LIN {X 0,Y 157.463,Z 192.851,A -85,B 0,C 180,E1 -23744.468,E2 -23744.468} C_VEL
LIN {X 0,Y 157.689,Z 192.84,A -85,B 0,C 180,E1 -23749.732,E2 -23749.732} C_VEL
LIN {X 0,Y 157.768,Z 192.832,A -85,B 0,C 180,E1 -23752.321,E2 -23752.321} C_VEL
LIN {X 0,Y 158.258,Z 192.764,A -85,B 0,C 180,E1 -23760.001,E2 -23760.001} C_VEL
LIN {X 0,Y 157.765,Z 192.822,A -85,B 0,C 180,E1 -23767.681,E2 -23767.681} C_VEL
LIN {X 0,Y 157.639,Z 192.844,A -85,B 0,C 180,E1 -23771.239,E2 -23771.239} C_VEL
LIN {X 0,Y 157.481,Z 192.867,A -85,B 0,C 180,E1 -23775.533,E2 -23775.533} C_VEL
LIN {X 0,Y 157.417,Z 192.875,A -85,B 0,C 180,E1 -23780.928,E2 -23780.928} C_VEL
LIN {X 0,Y 157.316,Z 192.89,A -85,B 0,C 180,E1 -23786.686,E2 -23786.686} C_VEL
LIN {X 0,Y 157.394,Z 192.935,A -85,B 0,C 180,E1 -23790.721,E2 -23790.721} C_VEL
LIN {X 0,Y 158.004,Z 196.792,A -85,B 0,C 180,E1 -23796.809,E2 -23796.809} C_VEL
LIN {X 0,Y 158.869,Z 201.219,A -85,B 0,C 180,E1 -23803.291,E2 -23803.291} C_VEL
LIN {X 0,Y 159.673,Z 205.204,A -85,B 0,C 180,E1 -23808.683,E2 -23808.683} C_VEL
LIN {X 0,Y 159.874,Z 206.674,A -85,B 0,C 180,E1 -23810.49,E2 -23810.49} C_VEL
LIN {X 0,Y 162.118,Z 215.988,A -85,B 0,C 180,E1 -23811.767,E2 -23811.767} C_VEL
LIN {X 0,Y 163.887,Z 229.522,A -85,B 0,C 180,E1 -23813.781,E2 -23813.781} C_VEL
LIN {X 0,Y 164.833,Z 241.541,A -85,B 0,C 180,E1 -23815.928,E2 -23815.928} C_VEL
LIN {X 0,Y 165.292,Z 252.413,A -85,B 0,C 180,E1 -23818.254,E2 -23818.254} C_VEL
LIN {X 0,Y 165.267,Z 263.527,A -85,B 0,C 180,E1 -23821.072,E2 -23821.072} C_VEL
LIN {X 0,Y 164.96,Z 269.314,A -85,B 0,C 180,E1 -23822.743,E2 -23822.743} C_VEL
LIN {X 0,Y 162.355,Z 278.226,A -85,B 0,C 180,E1 -23825.6,E2 -23825.6} C_VEL
LIN {X 0,Y 159.702,Z 287.461,A -85,B 0,C 180,E1 -23829.387,E2 -23829.387} C_VEL
LIN {X 0,Y 157.604,Z 294.658,A -85,B 0,C 180,E1 -23833.151,E2 -23833.151} C_VEL
LIN {X 0,Y 156.231,Z 300.428,A -85,B 0,C 180,E1 -23837.002,E2 -23837.002} C_VEL
LIN {X 0,Y 155.46,Z 304.944,A -85,B 0,C 180,E1 -23840.896,E2 -23840.896} C_VEL
LIN {X 0,Y 155.217,Z 308.458,A -85,B 0,C 180,E1 -23844.971,E2 -23844.971} C_VEL
LIN {X 0,Y 155.265,Z 310.005,A -85,B 0,C 180,E1 -23847.406,E2 -23847.406} C_VEL
LIN {X 0,Y 155.288,Z 311.229,A -85,B 0,C 180,E1 -23850,E2 -23850} C_VEL
LIN {X 0,Y 155.038,Z 312.3,A -85,B 0,C 180,E1 -23854.211,E2 -23854.211} C_VEL
LIN {X 0,Y 155.096,Z 312.412,A -85,B 0,C 180,E1 -23857.814,E2 -23857.814} C_VEL
LIN {X 0,Y 156.1,Z 311.257,A -85,B 0,C 180,E1 -23863.01,E2 -23863.01} C_VEL
LIN {X 0,Y 158.288,Z 308.643,A -85,B 0,C 180,E1 -23868.108,E2 -23868.108} C_VEL
LIN {X 0,Y 160.859,Z 305.623,A -85,B 0,C 180,E1 -23871.801,E2 -23871.801} C_VEL
LIN {X 0,Y 164.073,Z 301.657,A -85,B 0,C 180,E1 -23875.363,E2 -23875.363} C_VEL
LIN {X 0,Y 167.812,Z 296.682,A -85,B 0,C 180,E1 -23878.792,E2 -23878.792} C_VEL
LIN {X 0,Y 173.037,Z 289.457,A -85,B 0,C 180,E1 -23882.559,E2 -23882.559} C_VEL
LIN {X 0,Y 177.266,Z 283.144,A -85,B 0,C 180,E1 -23885.092,E2 -23885.092} C_VEL
LIN {X 0,Y 180.54,Z 275.915,A -85,B 0,C 180,E1 -23887.815,E2 -23887.815} C_VEL
LIN {X 0,Y 183.154,Z 267.778,A -85,B 0,C 180,E1 -23890.718,E2 -23890.718} C_VEL
LIN {X 0,Y 184.392,Z 262.401,A -85,B 0,C 180,E1 -23892.591,E2 -23892.591} C_VEL
LIN {X 0,Y 184.603,Z 260.007,A -85,B 0,C 180,E1 -23893.557,E2 -23893.557} C_VEL
LIN {X 0,Y 184.01,Z 257.051,A -85,B 0,C 180,E1 -23895.144,E2 -23895.144} C_VEL
LIN {X 0,Y 181.779,Z 253.248,A -85,B 0,C 180,E1 -23897.989,E2 -23897.989} C_VEL
LIN {X 0,Y 180.006,Z 250.364,A -85,B 0,C 180,E1 -23900.365,E2 -23900.365} C_VEL
LIN {X 0,Y 179.466,Z 248.695,A -85,B 0,C 180,E1 -23901.549,E2 -23901.549} C_VEL
LIN {X 0,Y 178.396,Z 243.679,A -85,B 0,C 180,E1 -23905.164,E2 -23905.164} C_VEL
LIN {X 0,Y 177.445,Z 239.467,A -85,B 0,C 180,E1 -23909.009,E2 -23909.009} C_VEL
LIN {X 0,Y 176.338,Z 236.354,A -85,B 0,C 180,E1 -23913.996,E2 -23913.996} C_VEL
LIN {X 0,Y 176.156,Z 235.271,A -85,B 0,C 180,E1 -23916.582,E2 -23916.582} C_VEL
LIN {X 0,Y 176.198,Z 234.757,A -85,B 0,C 180,E1 -23918.961,E2 -23918.961} C_VEL
LIN {X 0,Y 176.858,Z 234.904,A -85,B 0,C 180,E1 -23923.848,E2 -23923.848} C_VEL
LIN {X 0,Y 177.644,Z 235.267,A -85,B 0,C 180,E1 -23926.267,E2 -23926.267} C_VEL
LIN {X 0,Y 178.999,Z 238.295,A -85,B 0,C 180,E1 -23930.963,E2 -23930.963} C_VEL
LIN {X 0,Y 180.79,Z 242.663,A -85,B 0,C 180,E1 -23935.54,E2 -23935.54} C_VEL
LIN {X 0,Y 181.708,Z 247.304,A -85,B 0,C 180,E1 -23938.891,E2 -23938.891} C_VEL
LIN {X 0,Y 182.129,Z 251.884,A -85,B 0,C 180,E1 -23941.657,E2 -23941.657} C_VEL
LIN {X 0,Y 181.604,Z 258.398,A -85,B 0,C 180,E1 -23944.994,E2 -23944.994} C_VEL
LIN {X 0,Y 181.219,Z 260.675,A -85,B 0,C 180,E1 -23946.121,E2 -23946.121} C_VEL
LIN {X 0,Y 180.563,Z 262.357,A -85,B 0,C 180,E1 -23946.785,E2 -23946.785} C_VEL
LIN {X 0,Y 174.841,Z 270.868,A -85,B 0,C 180,E1 -23949.725,E2 -23949.725} C_VEL
LIN {X 0,Y 169.025,Z 278.432,A -85,B 0,C 180,E1 -23953.184,E2 -23953.184} C_VEL
LIN {X 0,Y 163.924,Z 284.316,A -85,B 0,C 180,E1 -23956.82,E2 -23956.82} C_VEL
LIN {X 0,Y 159.457,Z 288.794,A -85,B 0,C 180,E1 -23960.645,E2 -23960.645} C_VEL
LIN {X 0,Y 155.341,Z 292.384,A -85,B 0,C 180,E1 -23965.195,E2 -23965.195} C_VEL
LIN {X 0,Y 152.671,Z 294.266,A -85,B 0,C 180,E1 -23968.997,E2 -23968.997} C_VEL
LIN {X 0,Y 150.028,Z 295.433,A -85,B 0,C 180,E1 -23974.202,E2 -23974.202} C_VEL
LIN {X 0,Y 148.835,Z 295.324,A -85,B 0,C 180,E1 -23977.867,E2 -23977.867} C_VEL
LIN {X 0,Y 148.082,Z 294.5,A -85,B 0,C 180,E1 -23981.638,E2 -23981.638} C_VEL
LIN {X 0,Y 147.8,Z 292.89,A -85,B 0,C 180,E1 -23985.499,E2 -23985.499} C_VEL
LIN {X 0,Y 148.195,Z 289.33,A -85,B 0,C 180,E1 -23990.732,E2 -23990.732} C_VEL
LIN {X 0,Y 149.299,Z 284.523,A -85,B 0,C 180,E1 -23995.605,E2 -23995.605} C_VEL
LIN {X 0,Y 150.77,Z 278.971,A -85,B 0,C 180,E1 -23999.803,E2 -23999.803} C_VEL
LIN {X 0,Y 152.869,Z 271.595,A -85,B 0,C 180,E1 -24004.102,E2 -24004.102} C_VEL
LIN {X 0,Y 155.593,Z 262.734,A -85,B 0,C 180,E1 -24008.121,E2 -24008.121} C_VEL
LIN {X 0,Y 158.457,Z 252.842,A -85,B 0,C 180,E1 -24011.599,E2 -24011.599} C_VEL
LIN {X 0,Y 161.225,Z 242.566,A -85,B 0,C 180,E1 -24014.457,E2 -24014.457} C_VEL
LIN {X 0,Y 162.267,Z 237.854,A -85,B 0,C 180,E1 -24015.579,E2 -24015.579} C_VEL
LIN {X 0,Y 160.82,Z 227.521,A -85,B 0,C 180,E1 -24018.241,E2 -24018.241} C_VEL
LIN {X 0,Y 158.624,Z 216.159,A -85,B 0,C 180,E1 -24020.807,E2 -24020.807} C_VEL
LIN {X 0,Y 155.818,Z 206.445,A -85,B 0,C 180,E1 -24022.867,E2 -24022.867} C_VEL
LIN {X 0,Y 151.984,Z 197.063,A -85,B 0,C 180,E1 -24024.859,E2 -24024.859} C_VEL
LIN {X 0,Y 150.781,Z 194.317,A -85,B 0,C 180,E1 -24025.405,E2 -24025.405} C_VEL
LIN {X 0,Y 150.684,Z 193.719,A -85,B 0,C 180,E1 -24025.569,E2 -24025.569} C_VEL
LIN {X 0,Y 151.216,Z 193.647,A -85,B 0,C 180,E1 -24030,E2 -24030} C_VEL
LIN {X 0,Y 150.76,Z 193.71,A -85,B 0,C 180,E1 -24038.039,E2 -24038.039} C_VEL
LIN {X 0,Y 150.632,Z 193.719,A -85,B 0,C 180,E1 -24041.546,E2 -24041.546} C_VEL
LIN {X 0,Y 150.394,Z 193.752,A -85,B 0,C 180,E1 -24046.283,E2 -24046.283} C_VEL
LIN {X 0,Y 150.387,Z 193.756,A -85,B 0,C 180,E1 -24050.831,E2 -24050.831} C_VEL
LIN {X 0,Y 150.241,Z 193.761,A -85,B 0,C 180,E1 -24057.282,E2 -24057.282} C_VEL
LIN {X 0,Y 150.211,Z 193.775,A -85,B 0,C 180,E1 -24062.632,E2 -24062.632} C_VEL
LIN {X 0,Y 150.169,Z 193.766,A -85,B 0,C 180,E1 -24067.474,E2 -24067.474} C_VEL
LIN {X 0,Y 150.147,Z 193.782,A -85,B 0,C 180,E1 -24071.505,E2 -24071.505} C_VEL
LIN {X 0,Y 150.123,Z 193.777,A -85,B 0,C 180,E1 -24075.396,E2 -24075.396} C_VEL
LIN {X 0,Y 150.147,Z 193.764,A -85,B 0,C 180,E1 -24079.059,E2 -24079.059} C_VEL
LIN {X 0,Y 150.177,Z 193.775,A -85,B 0,C 180,E1 -24082.709,E2 -24082.709} C_VEL
LIN {X 0,Y 150.212,Z 193.768,A -85,B 0,C 180,E1 -24087.369,E2 -24087.369} C_VEL
LIN {X 0,Y 150.242,Z 193.753,A -85,B 0,C 180,E1 -24092.719,E2 -24092.719} C_VEL
LIN {X 0,Y 150.389,Z 193.749,A -85,B 0,C 180,E1 -24099.17,E2 -24099.17} C_VEL
LIN {X 0,Y 150.375,Z 193.735,A -85,B 0,C 180,E1 -24103.716,E2 -24103.716} C_VEL
LIN {X 0,Y 150.611,Z 193.721,A -85,B 0,C 180,E1 -24109.244,E2 -24109.244} C_VEL
LIN {X 0,Y 150.705,Z 193.713,A -85,B 0,C 180,E1 -24111.959,E2 -24111.959} C_VEL
LIN {X 0,Y 151.218,Z 193.64,A -85,B 0,C 180,E1 -24120.001,E2 -24120.001} C_VEL
LIN {X 0,Y 150.687,Z 193.701,A -85,B 0,C 180,E1 -24128.045,E2 -24128.045} C_VEL
LIN {X 0,Y 150.579,Z 193.724,A -85,B 0,C 180,E1 -24131.439,E2 -24131.439} C_VEL
LIN {X 0,Y 150.392,Z 193.746,A -85,B 0,C 180,E1 -24136.285,E2 -24136.285} C_VEL
LIN {X 0,Y 150.391,Z 193.75,A -85,B 0,C 180,E1 -24140.833,E2 -24140.833} C_VEL
LIN {X 0,Y 150.248,Z 193.772,A -85,B 0,C 180,E1 -24147.285,E2 -24147.285} C_VEL
LIN {X 0,Y 150.294,Z 193.83,A -85,B 0,C 180,E1 -24150.18,E2 -24150.18} C_VEL
LIN {X 0,Y 150.639,Z 196.137,A -85,B 0,C 180,E1 -24154.047,E2 -24154.047} C_VEL
LIN {X 0,Y 151.081,Z 198.423,A -85,B 0,C 180,E1 -24157.74,E2 -24157.74} C_VEL
LIN {X 0,Y 151.903,Z 202.558,A -85,B 0,C 180,E1 -24163.949,E2 -24163.949} C_VEL
LIN {X 0,Y 152.673,Z 206.336,A -85,B 0,C 180,E1 -24169.059,E2 -24169.059} C_VEL
LIN {X 0,Y 153.739,Z 209.669,A -85,B 0,C 180,E1 -24169.566,E2 -24169.566} C_VEL
LIN {X 0,Y 155.719,Z 217.222,A -85,B 0,C 180,E1 -24170.741,E2 -24170.741} C_VEL
LIN {X 0,Y 157.251,Z 229.909,A -85,B 0,C 180,E1 -24172.739,E2 -24172.739} C_VEL
LIN {X 0,Y 158.108,Z 241.252,A -85,B 0,C 180,E1 -24174.895,E2 -24174.895} C_VEL
LIN {X 0,Y 158.475,Z 252.458,A -85,B 0,C 180,E1 -24177.418,E2 -24177.418} C_VEL
LIN {X 0,Y 158.385,Z 263.687,A -85,B 0,C 180,E1 -24180.42,E2 -24180.42} C_VEL
LIN {X 0,Y 158.044,Z 269.421,A -85,B 0,C 180,E1 -24182.166,E2 -24182.166} C_VEL
LIN {X 0,Y 155.213,Z 278.695,A -85,B 0,C 180,E1 -24185.328,E2 -24185.328} C_VEL
LIN {X 0,Y 152.622,Z 287.374,A -85,B 0,C 180,E1 -24189.092,E2 -24189.092} C_VEL
LIN {X 0,Y 150.504,Z 294.512,A -85,B 0,C 180,E1 -24193.032,E2 -24193.032} C_VEL
LIN {X 0,Y 149.303,Z 299.333,A -85,B 0,C 180,E1 -24196.388,E2 -24196.388} C_VEL
LIN {X 0,Y 148.458,Z 303.997,A -85,B 0,C 180,E1 -24200.463,E2 -24200.463} C_VEL
LIN {X 0,Y 148.143,Z 307.892,A -85,B 0,C 180,E1 -24205.052,E2 -24205.052} C_VEL
LIN {X 0,Y 148.183,Z 309.302,A -85,B 0,C 180,E1 -24207.282,E2 -24207.282} C_VEL
LIN {X 0,Y 148.226,Z 310.592,A -85,B 0,C 180,E1 -24210,E2 -24210} C_VEL
LIN {X 0,Y 147.977,Z 311.743,A -85,B 0,C 180,E1 -24214.137,E2 -24214.137} C_VEL
LIN {X 0,Y 148.036,Z 311.979,A -85,B 0,C 180,E1 -24218.189,E2 -24218.189} C_VEL
LIN {X 0,Y 148.467,Z 311.676,A -85,B 0,C 180,E1 -24220.915,E2 -24220.915} C_VEL
LIN {X 0,Y 150.123,Z 309.924,A -85,B 0,C 180,E1 -24226.314,E2 -24226.314} C_VEL
LIN {X 0,Y 153.299,Z 306.7,A -85,B 0,C 180,E1 -24231.516,E2 -24231.516} C_VEL
LIN {X 0,Y 156.451,Z 303.214,A -85,B 0,C 180,E1 -24235.262,E2 -24235.262} C_VEL
LIN {X 0,Y 160.239,Z 298.763,A -85,B 0,C 180,E1 -24238.846,E2 -24238.846} C_VEL
LIN {X 0,Y 165.431,Z 292.227,A -85,B 0,C 180,E1 -24242.797,E2 -24242.797} C_VEL
LIN {X 0,Y 170.716,Z 285.201,A -85,B 0,C 180,E1 -24245.92,E2 -24245.92} C_VEL
LIN {X 0,Y 174.343,Z 278.487,A -85,B 0,C 180,E1 -24248.67,E2 -24248.67} C_VEL
LIN {X 0,Y 177.251,Z 270.999,A -85,B 0,C 180,E1 -24251.548,E2 -24251.548} C_VEL
LIN {X 0,Y 179.318,Z 263.592,A -85,B 0,C 180,E1 -24254.298,E2 -24254.298} C_VEL
LIN {X 0,Y 180.404,Z 258.267,A -85,B 0,C 180,E1 -24256.313,E2 -24256.313} C_VEL
LIN {X 0,Y 180.532,Z 255.172,A -85,B 0,C 180,E1 -24257.703,E2 -24257.703} C_VEL
LIN {X 0,Y 179.466,Z 248.695,A -85,B 0,C 180,E1 -24261.549,E2 -24261.549} C_VEL
LIN {X 0,Y 178.564,Z 246.71,A -85,B 0,C 180,E1 -24263.301,E2 -24263.301} C_VEL
LIN {X 0,Y 177.18,Z 245.666,A -85,B 0,C 180,E1 -24265.131,E2 -24265.131} C_VEL
LIN {X 0,Y 173.518,Z 244.495,A -85,B 0,C 180,E1 -24270.247,E2 -24270.247} C_VEL
LIN {X 0,Y 173.088,Z 243.904,A -85,B 0,C 180,E1 -24271.56,E2 -24271.56} C_VEL
LIN {X 0,Y 172.619,Z 241.728,A -85,B 0,C 180,E1 -24275.974,E2 -24275.974} C_VEL
LIN {X 0,Y 172.701,Z 240.889,A -85,B 0,C 180,E1 -24279.388,E2 -24279.388} C_VEL
LIN {X 0,Y 173.866,Z 241.276,A -85,B 0,C 180,E1 -24285.963,E2 -24285.963} C_VEL
LIN {X 0,Y 174.98,Z 244.09,A -85,B 0,C 180,E1 -24290.754,E2 -24290.754} C_VEL
LIN {X 0,Y 176.319,Z 248.343,A -85,B 0,C 180,E1 -24295.426,E2 -24295.426} C_VEL
LIN {X 0,Y 176.829,Z 252.868,A -85,B 0,C 180,E1 -24298.86,E2 -24298.86} C_VEL
LIN {X 0,Y 176.825,Z 256.432,A -85,B 0,C 180,E1 -24301.138,E2 -24301.138} C_VEL
LIN {X 0,Y 175.838,Z 262.639,A -85,B 0,C 180,E1 -24304.584,E2 -24304.584} C_VEL
LIN {X 0,Y 175.509,Z 263.762,A -85,B 0,C 180,E1 -24305.168,E2 -24305.168} C_VEL
LIN {X 0,Y 170.267,Z 271.258,A -85,B 0,C 180,E1 -24307.845,E2 -24307.845} C_VEL
LIN {X 0,Y 164.664,Z 278.164,A -85,B 0,C 180,E1 -24310.986,E2 -24310.986} C_VEL
LIN {X 0,Y 159.568,Z 283.694,A -85,B 0,C 180,E1 -24314.309,E2 -24314.309} C_VEL
LIN {X 0,Y 154.119,Z 288.91,A -85,B 0,C 180,E1 -24318.614,E2 -24318.614} C_VEL
LIN {X 0,Y 149.289,Z 292.805,A -85,B 0,C 180,E1 -24323.586,E2 -24323.586} C_VEL
LIN {X 0,Y 145.486,Z 295.163,A -85,B 0,C 180,E1 -24328.884,E2 -24328.884} C_VEL
LIN {X 0,Y 143.17,Z 295.928,A -85,B 0,C 180,E1 -24333.434,E2 -24333.434} C_VEL
LIN {X 0,Y 141.796,Z 295.721,A -85,B 0,C 180,E1 -24337.53,E2 -24337.53} C_VEL
LIN {X 0,Y 140.981,Z 294.721,A -85,B 0,C 180,E1 -24341.602,E2 -24341.602} C_VEL
LIN {X 0,Y 140.698,Z 292.969,A -85,B 0,C 180,E1 -24345.627,E2 -24345.627} C_VEL
LIN {X 0,Y 141.18,Z 289.173,A -85,B 0,C 180,E1 -24351.236,E2 -24351.236} C_VEL
LIN {X 0,Y 142.094,Z 285.274,A -85,B 0,C 180,E1 -24355.309,E2 -24355.309} C_VEL
LIN {X 0,Y 143.619,Z 279.574,A -85,B 0,C 180,E1 -24359.895,E2 -24359.895} C_VEL
LIN {X 0,Y 145.721,Z 272.467,A -85,B 0,C 180,E1 -24364.274,E2 -24364.274} C_VEL
LIN {X 0,Y 148.334,Z 264.163,A -85,B 0,C 180,E1 -24368.28,E2 -24368.28} C_VEL
LIN {X 0,Y 151.104,Z 255.196,A -85,B 0,C 180,E1 -24371.702,E2 -24371.702} C_VEL
LIN {X 0,Y 154.096,Z 244.667,A -85,B 0,C 180,E1 -24374.857,E2 -24374.857} C_VEL
LIN {X 0,Y 155.494,Z 239.051,A -85,B 0,C 180,E1 -24376.273,E2 -24376.273} C_VEL
LIN {X 0,Y 154.078,Z 228.523,A -85,B 0,C 180,E1 -24379.154,E2 -24379.154} C_VEL
LIN {X 0,Y 152.028,Z 217.496,A -85,B 0,C 180,E1 -24381.816,E2 -24381.816} C_VEL
LIN {X 0,Y 148.861,Z 206.895,A -85,B 0,C 180,E1 -24384.242,E2 -24384.242} C_VEL
LIN {X 0,Y 143.883,Z 195.26,A -85,B 0,C 180,E1 -24386.863,E2 -24386.863} C_VEL
LIN {X 0,Y 143.794,Z 194.572,A -85,B 0,C 180,E1 -24387.005,E2 -24387.005} C_VEL
LIN {X 0,Y 144.174,Z 194.524,A -85,B 0,C 180,E1 -24390,E2 -24390} C_VEL
LIN {X 0,Y 143.682,Z 194.59,A -85,B 0,C 180,E1 -24398.438,E2 -24398.438} C_VEL
LIN {X 0,Y 143.568,Z 194.6,A -85,B 0,C 180,E1 -24401.757,E2 -24401.757} C_VEL
LIN {X 0,Y 143.332,Z 194.629,A -85,B 0,C 180,E1 -24407.109,E2 -24407.109} C_VEL
LIN {X 0,Y 143.308,Z 194.64,A -85,B 0,C 180,E1 -24411.29,E2 -24411.29} C_VEL
LIN {X 0,Y 143.187,Z 194.644,A -85,B 0,C 180,E1 -24417.937,E2 -24417.937} C_VEL
LIN {X 0,Y 143.14,Z 194.652,A -85,B 0,C 180,E1 -24423.42,E2 -24423.42} C_VEL
LIN {X 0,Y 143.058,Z 194.662,A -85,B 0,C 180,E1 -24429.691,E2 -24429.691} C_VEL
LIN {X 0,Y 143.053,Z 194.664,A -85,B 0,C 180,E1 -24433.456,E2 -24433.456} C_VEL
LIN {X 0,Y 143.062,Z 194.646,A -85,B 0,C 180,E1 -24437.466,E2 -24437.466} C_VEL
LIN {X 0,Y 143.075,Z 194.658,A -85,B 0,C 180,E1 -24441.807,E2 -24441.807} C_VEL
LIN {X 0,Y 143.179,Z 194.644,A -85,B 0,C 180,E1 -24447.322,E2 -24447.322} C_VEL
LIN {X 0,Y 143.188,Z 194.629,A -85,B 0,C 180,E1 -24452.064,E2 -24452.064} C_VEL
LIN {X 0,Y 143.31,Z 194.632,A -85,B 0,C 180,E1 -24458.712,E2 -24458.712} C_VEL
LIN {X 0,Y 143.319,Z 194.616,A -85,B 0,C 180,E1 -24462.89,E2 -24462.89} C_VEL
LIN {X 0,Y 143.537,Z 194.602,A -85,B 0,C 180,E1 -24468.707,E2 -24468.707} C_VEL
LIN {X 0,Y 143.627,Z 194.594,A -85,B 0,C 180,E1 -24471.56,E2 -24471.56} C_VEL
LIN {X 0,Y 144.177,Z 194.517,A -85,B 0,C 180,E1 -24480.001,E2 -24480.001} C_VEL
LIN {X 0,Y 143.612,Z 194.581,A -85,B 0,C 180,E1 -24488.444,E2 -24488.444} C_VEL
LIN {X 0,Y 143.508,Z 194.605,A -85,B 0,C 180,E1 -24491.635,E2 -24491.635} C_VEL
LIN {X 0,Y 143.332,Z 194.623,A -85,B 0,C 180,E1 -24497.111,E2 -24497.111} C_VEL
LIN {X 0,Y 143.313,Z 194.633,A -85,B 0,C 180,E1 -24501.291,E2 -24501.291} C_VEL
LIN {X 0,Y 143.197,Z 194.65,A -85,B 0,C 180,E1 -24507.942,E2 -24507.942} C_VEL
LIN {X 0,Y 143.243,Z 194.821,A -85,B 0,C 180,E1 -24509.788,E2 -24509.788} C_VEL
LIN {X 0,Y 143.595,Z 197.022,A -85,B 0,C 180,E1 -24513.692,E2 -24513.692} C_VEL
LIN {X 0,Y 144.2,Z 200.417,A -85,B 0,C 180,E1 -24519.317,E2 -24519.317} C_VEL
LIN {X 0,Y 144.958,Z 203.91,A -85,B 0,C 180,E1 -24524.757,E2 -24524.757} C_VEL
LIN {X 0,Y 145.352,Z 205.798,A -85,B 0,C 180,E1 -24527.427,E2 -24527.427} C_VEL
LIN {X 0,Y 146.418,Z 209.084,A -85,B 0,C 180,E1 -24527.975,E2 -24527.975} C_VEL
LIN {X 0,Y 148.932,Z 216.839,A -85,B 0,C 180,E1 -24529.38,E2 -24529.38} C_VEL
LIN {X 0,Y 150.389,Z 227.72,A -85,B 0,C 180,E1 -24531.203,E2 -24531.203} C_VEL
LIN {X 0,Y 151.367,Z 240.552,A -85,B 0,C 180,E1 -24533.702,E2 -24533.702} C_VEL
LIN {X 0,Y 151.654,Z 252.603,A -85,B 0,C 180,E1 -24536.531,E2 -24536.531} C_VEL
LIN {X 0,Y 151.507,Z 263.838,A -85,B 0,C 180,E1 -24539.705,E2 -24539.705} C_VEL
LIN {X 0,Y 151.128,Z 269.498,A -85,B 0,C 180,E1 -24541.533,E2 -24541.533} C_VEL
LIN {X 0,Y 148.301,Z 278.483,A -85,B 0,C 180,E1 -24544.754,E2 -24544.754} C_VEL
LIN {X 0,Y 145.55,Z 287.287,A -85,B 0,C 180,E1 -24548.769,E2 -24548.769} C_VEL
LIN {X 0,Y 143.382,Z 294.353,A -85,B 0,C 180,E1 -24552.897,E2 -24552.897} C_VEL
LIN {X 0,Y 142.005,Z 299.983,A -85,B 0,C 180,E1 -24557.132,E2 -24557.132} C_VEL
LIN {X 0,Y 141.257,Z 304.382,A -85,B 0,C 180,E1 -24561.416,E2 -24561.416} C_VEL
LIN {X 0,Y 141.084,Z 307.251,A -85,B 0,C 180,E1 -24565.075,E2 -24565.075} C_VEL
LIN {X 0,Y 141.128,Z 308.534,A -85,B 0,C 180,E1 -24567.146,E2 -24567.146} C_VEL
LIN {X 0,Y 141.164,Z 309.934,A -85,B 0,C 180,E1 -24570,E2 -24570} C_VEL
LIN {X 0,Y 140.907,Z 311.1,A -85,B 0,C 180,E1 -24574.003,E2 -24574.003} C_VEL
LIN {X 0,Y 141,Z 311.51,A -85,B 0,C 180,E1 -24578.6,E2 -24578.6} C_VEL
LIN {X 0,Y 142.218,Z 310.703,A -85,B 0,C 180,E1 -24584.306,E2 -24584.306} C_VEL
LIN {X 0,Y 144.816,Z 308.377,A -85,B 0,C 180,E1 -24589.86,E2 -24589.86} C_VEL
LIN {X 0,Y 148.815,Z 304.56,A -85,B 0,C 180,E1 -24595.154,E2 -24595.154} C_VEL
LIN {X 0,Y 153.011,Z 300.216,A -85,B 0,C 180,E1 -24599.224,E2 -24599.224} C_VEL
LIN {X 0,Y 158.696,Z 293.721,A -85,B 0,C 180,E1 -24603.613,E2 -24603.613} C_VEL
LIN {X 0,Y 165.058,Z 286.003,A -85,B 0,C 180,E1 -24607.356,E2 -24607.356} C_VEL
LIN {X 0,Y 168.848,Z 279.49,A -85,B 0,C 180,E1 -24610.178,E2 -24610.178} C_VEL
LIN {X 0,Y 172.11,Z 271.972,A -85,B 0,C 180,E1 -24613.263,E2 -24613.263} C_VEL
LIN {X 0,Y 174.629,Z 264.127,A -85,B 0,C 180,E1 -24616.421,E2 -24616.421} C_VEL
LIN {X 0,Y 175.375,Z 260.442,A -85,B 0,C 180,E1 -24618.008,E2 -24618.008} C_VEL
LIN {X 0,Y 175.217,Z 256.896,A -85,B 0,C 180,E1 -24620.075,E2 -24620.075} C_VEL
LIN {X 0,Y 174.497,Z 251.735,A -85,B 0,C 180,E1 -24623.661,E2 -24623.661} C_VEL
LIN {X 0,Y 174.207,Z 249.25,A -85,B 0,C 180,E1 -24625.61,E2 -24625.61} C_VEL
LIN {X 0,Y 173.518,Z 245.174,A -85,B 0,C 180,E1 -24629.582,E2 -24629.582} C_VEL
LIN {X 0,Y 173.088,Z 243.904,A -85,B 0,C 180,E1 -24631.56,E2 -24631.56} C_VEL
LIN {X 0,Y 172.418,Z 243.446,A -85,B 0,C 180,E1 -24633.498,E2 -24633.498} C_VEL
LIN {X 0,Y 171.387,Z 243.951,A -85,B 0,C 180,E1 -24635.443,E2 -24635.443} C_VEL
LIN {X 0,Y 169.075,Z 246.601,A -85,B 0,C 180,E1 -24640.721,E2 -24640.721} C_VEL
LIN {X 0,Y 169.057,Z 246.837,A -85,B 0,C 180,E1 -24642.079,E2 -24642.079} C_VEL
LIN {X 0,Y 169.789,Z 247.129,A -85,B 0,C 180,E1 -24645.619,E2 -24645.619} C_VEL
LIN {X 0,Y 170.2,Z 248.233,A -85,B 0,C 180,E1 -24648.084,E2 -24648.084} C_VEL
LIN {X 0,Y 170.735,Z 250.124,A -85,B 0,C 180,E1 -24651.087,E2 -24651.087} C_VEL
LIN {X 0,Y 171.41,Z 252.624,A -85,B 0,C 180,E1 -24654.115,E2 -24654.115} C_VEL
LIN {X 0,Y 171.632,Z 254.68,A -85,B 0,C 180,E1 -24656.08,E2 -24656.08} C_VEL
LIN {X 0,Y 171.675,Z 258.187,A -85,B 0,C 180,E1 -24658.826,E2 -24658.826} C_VEL
LIN {X 0,Y 171.168,Z 261.755,A -85,B 0,C 180,E1 -24661.175,E2 -24661.175} C_VEL
LIN {X 0,Y 170.4,Z 265.129,A -85,B 0,C 180,E1 -24663.213,E2 -24663.213} C_VEL
LIN {X 0,Y 169.808,Z 266.619,A -85,B 0,C 180,E1 -24663.986,E2 -24663.986} C_VEL
LIN {X 0,Y 164.228,Z 273.737,A -85,B 0,C 180,E1 -24666.698,E2 -24666.698} C_VEL
LIN {X 0,Y 157.296,Z 281.374,A -85,B 0,C 180,E1 -24670.587,E2 -24670.587} C_VEL
LIN {X 0,Y 152.138,Z 286.337,A -85,B 0,C 180,E1 -24674.046,E2 -24674.046} C_VEL
LIN {X 0,Y 147.543,Z 290.192,A -85,B 0,C 180,E1 -24677.696,E2 -24677.696} C_VEL
LIN {X 0,Y 143.596,Z 293.069,A -85,B 0,C 180,E1 -24681.577,E2 -24681.577} C_VEL
LIN {X 0,Y 139.393,Z 295.499,A -85,B 0,C 180,E1 -24686.984,E2 -24686.984} C_VEL
LIN {X 0,Y 137.177,Z 296.265,A -85,B 0,C 180,E1 -24690.817,E2 -24690.817} C_VEL
LIN {X 0,Y 135.477,Z 296.369,A -85,B 0,C 180,E1 -24694.793,E2 -24694.793} C_VEL
LIN {X 0,Y 134.361,Z 295.731,A -85,B 0,C 180,E1 -24698.877,E2 -24698.877} C_VEL
LIN {X 0,Y 133.714,Z 294.322,A -85,B 0,C 180,E1 -24703.098,E2 -24703.098} C_VEL
LIN {X 0,Y 133.638,Z 292.089,A -85,B 0,C 180,E1 -24707.411,E2 -24707.411} C_VEL
LIN {X 0,Y 134.171,Z 288.934,A -85,B 0,C 180,E1 -24711.784,E2 -24711.784} C_VEL
LIN {X 0,Y 135.211,Z 284.637,A -85,B 0,C 180,E1 -24716.265,E2 -24716.265} C_VEL
LIN {X 0,Y 136.836,Z 278.969,A -85,B 0,C 180,E1 -24720.822,E2 -24720.822} C_VEL
LIN {X 0,Y 139.097,Z 271.612,A -85,B 0,C 180,E1 -24725.428,E2 -24725.428} C_VEL
LIN {X 0,Y 142.069,Z 262.667,A -85,B 0,C 180,E1 -24729.739,E2 -24729.739} C_VEL
LIN {X 0,Y 145.129,Z 252.82,A -85,B 0,C 180,E1 -24733.429,E2 -24733.429} C_VEL
LIN {X 0,Y 147.905,Z 243.295,A -85,B 0,C 180,E1 -24736.255,E2 -24736.255} C_VEL
LIN {X 0,Y 148.7,Z 240.276,A -85,B 0,C 180,E1 -24737.026,E2 -24737.026} C_VEL
LIN {X 0,Y 147.486,Z 230.146,A -85,B 0,C 180,E1 -24739.97,E2 -24739.97} C_VEL
LIN {X 0,Y 145.595,Z 219.495,A -85,B 0,C 180,E1 -24742.72,E2 -24742.72} C_VEL
LIN {X 0,Y 142.731,Z 209.764,A -85,B 0,C 180,E1 -24745.127,E2 -24745.127} C_VEL
LIN {X 0,Y 137.226,Z 196.899,A -85,B 0,C 180,E1 -24748.349,E2 -24748.349} C_VEL
LIN {X 0,Y 136.93,Z 195.43,A -85,B 0,C 180,E1 -24748.713,E2 -24748.713} C_VEL
LIN {X 0,Y 137.13,Z 195.401,A -85,B 0,C 180,E1 -24749.999,E2 -24749.999} C_VEL
LIN {X 0,Y 136.606,Z 195.472,A -85,B 0,C 180,E1 -24758.878,E2 -24758.878} C_VEL
LIN {X 0,Y 136.49,Z 195.483,A -85,B 0,C 180,E1 -24761.959,E2 -24761.959} C_VEL
LIN {X 0,Y 136.271,Z 195.506,A -85,B 0,C 180,E1 -24768.025,E2 -24768.025} C_VEL
LIN {X 0,Y 136.224,Z 195.523,A -85,B 0,C 180,E1 -24771.78,E2 -24771.78} C_VEL
LIN {X 0,Y 136.097,Z 195.529,A -85,B 0,C 180,E1 -24778.616,E2 -24778.616} C_VEL
LIN {X 0,Y 136.039,Z 195.53,A -85,B 0,C 180,E1 -24784.63,E2 -24784.63} C_VEL
LIN {X 0,Y 136.028,Z 195.534,A -85,B 0,C 180,E1 -24789.199,E2 -24789.199} C_VEL
LIN {X 0,Y 135.995,Z 195.542,A -85,B 0,C 180,E1 -24793.658,E2 -24793.658} C_VEL
LIN {X 0,Y 136.002,Z 195.523,A -85,B 0,C 180,E1 -24797.797,E2 -24797.797} C_VEL
LIN {X 0,Y 136.025,Z 195.536,A -85,B 0,C 180,E1 -24801.685,E2 -24801.685} C_VEL
LIN {X 0,Y 136.082,Z 195.532,A -85,B 0,C 180,E1 -24805.722,E2 -24805.722} C_VEL
LIN {X 0,Y 136.145,Z 195.506,A -85,B 0,C 180,E1 -24812.318,E2 -24812.318} C_VEL
LIN {X 0,Y 136.277,Z 195.508,A -85,B 0,C 180,E1 -24818.84,E2 -24818.84} C_VEL
LIN {X 0,Y 136.275,Z 195.488,A -85,B 0,C 180,E1 -24825.058,E2 -24825.058} C_VEL
LIN {X 0,Y 136.444,Z 195.482,A -85,B 0,C 180,E1 -24828.139,E2 -24828.139} C_VEL
LIN {X 0,Y 136.552,Z 195.475,A -85,B 0,C 180,E1 -24831.119,E2 -24831.119} C_VEL
LIN {X 0,Y 137.133,Z 195.394,A -85,B 0,C 180,E1 -24840.002,E2 -24840.002} C_VEL
LIN {X 0,Y 136.541,Z 195.461,A -85,B 0,C 180,E1 -24848.884,E2 -24848.884} C_VEL
LIN {X 0,Y 136.459,Z 195.484,A -85,B 0,C 180,E1 -24851.89,E2 -24851.89} C_VEL
LIN {X 0,Y 136.273,Z 195.5,A -85,B 0,C 180,E1 -24858.027,E2 -24858.027} C_VEL
LIN {X 0,Y 136.229,Z 195.517,A -85,B 0,C 180,E1 -24861.781,E2 -24861.781} C_VEL
LIN {X 0,Y 136.191,Z 195.604,A -85,B 0,C 180,E1 -24869.034,E2 -24869.034} C_VEL
LIN {X 0,Y 136.416,Z 196.642,A -85,B 0,C 180,E1 -24871.012,E2 -24871.012} C_VEL
LIN {X 0,Y 137.001,Z 200.577,A -85,B 0,C 180,E1 -24877.996,E2 -24877.996} C_VEL
LIN {X 0,Y 137.85,Z 204.508,A -85,B 0,C 180,E1 -24884.459,E2 -24884.459} C_VEL
LIN {X 0,Y 138.008,Z 205.238,A -85,B 0,C 180,E1 -24885.607,E2 -24885.607} C_VEL
LIN {X 0,Y 139.182,Z 208.778,A -85,B 0,C 180,E1 -24886.281,E2 -24886.281} C_VEL
LIN {X 0,Y 142.306,Z 217.428,A -85,B 0,C 180,E1 -24888.033,E2 -24888.033} C_VEL
LIN {X 0,Y 143.53,Z 224.763,A -85,B 0,C 180,E1 -24889.377,E2 -24889.377} C_VEL
LIN {X 0,Y 144.547,Z 238.079,A -85,B 0,C 180,E1 -24892.043,E2 -24892.043} C_VEL
LIN {X 0,Y 144.867,Z 250.418,A -85,B 0,C 180,E1 -24894.987,E2 -24894.987} C_VEL
LIN {X 0,Y 144.699,Z 261.323,A -85,B 0,C 180,E1 -24898.117,E2 -24898.117} C_VEL
LIN {X 0,Y 144.24,Z 269.473,A -85,B 0,C 180,E1 -24900.841,E2 -24900.841} C_VEL
LIN {X 0,Y 141.33,Z 278.38,A -85,B 0,C 180,E1 -24904.208,E2 -24904.208} C_VEL
LIN {X 0,Y 138.514,Z 287.117,A -85,B 0,C 180,E1 -24908.417,E2 -24908.417} C_VEL
LIN {X 0,Y 136.298,Z 294.108,A -85,B 0,C 180,E1 -24912.754,E2 -24912.754} C_VEL
LIN {X 0,Y 134.744,Z 300.488,A -85,B 0,C 180,E1 -24917.958,E2 -24917.958} C_VEL
LIN {X 0,Y 134.104,Z 304.658,A -85,B 0,C 180,E1 -24922.472,E2 -24922.472} C_VEL
LIN {X 0,Y 134.073,Z 307.739,A -85,B 0,C 180,E1 -24926.996,E2 -24926.996} C_VEL
LIN {X 0,Y 134.103,Z 309.215,A -85,B 0,C 180,E1 -24930.001,E2 -24930.001} C_VEL
LIN {X 0,Y 133.86,Z 310.458,A -85,B 0,C 180,E1 -24933.994,E2 -24933.994} C_VEL
LIN {X 0,Y 133.984,Z 311.04,A -85,B 0,C 180,E1 -24939.054,E2 -24939.054} C_VEL
LIN {X 0,Y 135.322,Z 310.381,A -85,B 0,C 180,E1 -24945.051,E2 -24945.051} C_VEL
LIN {X 0,Y 136.48,Z 309.514,A -85,B 0,C 180,E1 -24947.998,E2 -24947.998} C_VEL
LIN {X 0,Y 140.106,Z 306.623,A -85,B 0,C 180,E1 -24953.66,E2 -24953.66} C_VEL
LIN {X 0,Y 145.074,Z 302.197,A -85,B 0,C 180,E1 -24958.976,E2 -24958.976} C_VEL
LIN {X 0,Y 149.506,Z 297.767,A -85,B 0,C 180,E1 -24962.725,E2 -24962.725} C_VEL
LIN {X 0,Y 154.673,Z 292.273,A -85,B 0,C 180,E1 -24966.207,E2 -24966.207} C_VEL
LIN {X 0,Y 159.499,Z 286.754,A -85,B 0,C 180,E1 -24968.896,E2 -24968.896} C_VEL
LIN {X 0,Y 163.492,Z 280.54,A -85,B 0,C 180,E1 -24971.782,E2 -24971.782} C_VEL
LIN {X 0,Y 166.988,Z 273.434,A -85,B 0,C 180,E1 -24974.916,E2 -24974.916} C_VEL
LIN {X 0,Y 169.74,Z 265.88,A -85,B 0,C 180,E1 -24978.184,E2 -24978.184} C_VEL
LIN {X 0,Y 170.239,Z 263.38,A -85,B 0,C 180,E1 -24979.475,E2 -24979.475} C_VEL
LIN {X 0,Y 170.017,Z 258.779,A -85,B 0,C 180,E1 -24982.669,E2 -24982.669} C_VEL
LIN {X 0,Y 169.734,Z 254.814,A -85,B 0,C 180,E1 -24985.907,E2 -24985.907} C_VEL
LIN {X 0,Y 169.229,Z 250.333,A -85,B 0,C 180,E1 -24990.707,E2 -24990.707} C_VEL
LIN {X 0,Y 168.744,Z 247.579,A -85,B 0,C 180,E1 -24996.389,E2 -24996.389} C_VEL
LIN {X 0,Y 168.923,Z 246.797,A -85,B 0,C 180,E1 -25000.558,E2 -25000.558} C_VEL
LIN {X 0,Y 169.057,Z 246.837,A -85,B 0,C 180,E1 -25002.079,E2 -25002.079} C_VEL
LIN {X 0,Y 168.963,Z 247.578,A -85,B 0,C 180,E1 -25004.062,E2 -25004.062} C_VEL
LIN {X 0,Y 168.365,Z 249.32,A -85,B 0,C 180,E1 -25005.983,E2 -25005.983} C_VEL
LIN {X 0,Y 166.357,Z 255.44,A -85,B 0,C 180,E1 -25011.064,E2 -25011.064} C_VEL
LIN {X 0,Y 166.35,Z 256.606,A -85,B 0,C 180,E1 -25012.398,E2 -25012.398} C_VEL
LIN {X 0,Y 166.582,Z 259.007,A -85,B 0,C 180,E1 -25015.158,E2 -25015.158} C_VEL
LIN {X 0,Y 166.221,Z 263.288,A -85,B 0,C 180,E1 -25018.787,E2 -25018.787} C_VEL
LIN {X 0,Y 165.276,Z 266.795,A -85,B 0,C 180,E1 -25021.217,E2 -25021.217} C_VEL
LIN {X 0,Y 164.571,Z 268.728,A -85,B 0,C 180,E1 -25022.446,E2 -25022.446} C_VEL
LIN {X 0,Y 157.383,Z 277.09,A -85,B 0,C 180,E1 -25025.921,E2 -25025.921} C_VEL
LIN {X 0,Y 151.797,Z 282.643,A -85,B 0,C 180,E1 -25028.995,E2 -25028.995} C_VEL
LIN {X 0,Y 146.691,Z 287.124,A -85,B 0,C 180,E1 -25032.286,E2 -25032.286} C_VEL
LIN {X 0,Y 142.069,Z 290.709,A -85,B 0,C 180,E1 -25035.786,E2 -25035.786} C_VEL
LIN {X 0,Y 136.514,Z 294.341,A -85,B 0,C 180,E1 -25041.121,E2 -25041.121} C_VEL
LIN {X 0,Y 132.796,Z 296.132,A -85,B 0,C 180,E1 -25045.881,E2 -25045.881} C_VEL
LIN {X 0,Y 130.23,Z 296.829,A -85,B 0,C 180,E1 -25050.291,E2 -25050.291} C_VEL
LIN {X 0,Y 128.331,Z 296.711,A -85,B 0,C 180,E1 -25054.766,E2 -25054.766} C_VEL
LIN {X 0,Y 127.144,Z 295.806,A -85,B 0,C 180,E1 -25059.297,E2 -25059.297} C_VEL
LIN {X 0,Y 126.563,Z 294.155,A -85,B 0,C 180,E1 -25063.789,E2 -25063.789} C_VEL
LIN {X 0,Y 126.612,Z 291.723,A -85,B 0,C 180,E1 -25068.232,E2 -25068.232} C_VEL
LIN {X 0,Y 127.186,Z 288.507,A -85,B 0,C 180,E1 -25072.566,E2 -25072.566} C_VEL
LIN {X 0,Y 128.505,Z 283.491,A -85,B 0,C 180,E1 -25077.719,E2 -25077.719} C_VEL
LIN {X 0,Y 130.435,Z 277.053,A -85,B 0,C 180,E1 -25082.742,E2 -25082.742} C_VEL
LIN {X 0,Y 133.028,Z 269.168,A -85,B 0,C 180,E1 -25087.478,E2 -25087.478} C_VEL
LIN {X 0,Y 135.971,Z 260.663,A -85,B 0,C 180,E1 -25091.472,E2 -25091.472} C_VEL
LIN {X 0,Y 139.029,Z 251.238,A -85,B 0,C 180,E1 -25094.963,E2 -25094.963} C_VEL
LIN {X 0,Y 141.896,Z 241.44,A -85,B 0,C 180,E1 -25097.848,E2 -25097.848} C_VEL
LIN {X 0,Y 140.961,Z 232.247,A -85,B 0,C 180,E1 -25100.674,E2 -25100.674} C_VEL
LIN {X 0,Y 139.311,Z 222.169,A -85,B 0,C 180,E1 -25103.482,E2 -25103.482} C_VEL
LIN {X 0,Y 136.886,Z 213.317,A -85,B 0,C 180,E1 -25105.88,E2 -25105.88} C_VEL
LIN {X 0,Y 131.997,Z 201.561,A -85,B 0,C 180,E1 -25109.108,E2 -25109.108} C_VEL
LIN {X 0,Y 130.002,Z 196.287,A -85,B 0,C 180,E1 -25110.483,E2 -25110.483} C_VEL
LIN {X 0,Y 129.528,Z 196.35,A -85,B 0,C 180,E1 -25119.368,E2 -25119.368} C_VEL
LIN {X 0,Y 129.392,Z 196.372,A -85,B 0,C 180,E1 -25122.548,E2 -25122.548} C_VEL
LIN {X 0,Y 129.183,Z 196.392,A -85,B 0,C 180,E1 -25129.051,E2 -25129.051} C_VEL
LIN {X 0,Y 129.133,Z 196.405,A -85,B 0,C 180,E1 -25132.393,E2 -25132.393} C_VEL
LIN {X 0,Y 129.013,Z 196.414,A -85,B 0,C 180,E1 -25139.358,E2 -25139.358} C_VEL
LIN {X 0,Y 128.955,Z 196.408,A -85,B 0,C 180,E1 -25145.168,E2 -25145.168} C_VEL
LIN {X 0,Y 128.931,Z 196.423,A -85,B 0,C 180,E1 -25150.852,E2 -25150.852} C_VEL
LIN {X 0,Y 128.919,Z 196.419,A -85,B 0,C 180,E1 -25155.128,E2 -25155.128} C_VEL
LIN {X 0,Y 128.939,Z 196.408,A -85,B 0,C 180,E1 -25159.737,E2 -25159.737} C_VEL
LIN {X 0,Y 128.979,Z 196.419,A -85,B 0,C 180,E1 -25164.819,E2 -25164.819} C_VEL
LIN {X 0,Y 129.014,Z 196.391,A -85,B 0,C 180,E1 -25170.644,E2 -25170.644} C_VEL
LIN {X 0,Y 129.135,Z 196.398,A -85,B 0,C 180,E1 -25177.608,E2 -25177.608} C_VEL
LIN {X 0,Y 129.178,Z 196.386,A -85,B 0,C 180,E1 -25180.949,E2 -25180.949} C_VEL
LIN {X 0,Y 129.367,Z 196.363,A -85,B 0,C 180,E1 -25187.922,E2 -25187.922} C_VEL
LIN {X 0,Y 129.477,Z 196.357,A -85,B 0,C 180,E1 -25190.63,E2 -25190.63} C_VEL
LIN {X 0,Y 130.088,Z 196.271,A -85,B 0,C 180,E1 -25200.002,E2 -25200.002} C_VEL
LIN {X 0,Y 129.472,Z 196.342,A -85,B 0,C 180,E1 -25209.374,E2 -25209.374} C_VEL
LIN {X 0,Y 129.353,Z 196.372,A -85,B 0,C 180,E1 -25212.554,E2 -25212.554} C_VEL
LIN {X 0,Y 129.186,Z 196.384,A -85,B 0,C 180,E1 -25219.053,E2 -25219.053} C_VEL
LIN {X 0,Y 129.137,Z 196.399,A -85,B 0,C 180,E1 -25222.395,E2 -25222.395} C_VEL
LIN {X 0,Y 129.148,Z 196.497,A -85,B 0,C 180,E1 -25228.437,E2 -25228.437} C_VEL
LIN {X 0,Y 129.475,Z 198.752,A -85,B 0,C 180,E1 -25232.877,E2 -25232.877} C_VEL
LIN {X 0,Y 130.003,Z 201.779,A -85,B 0,C 180,E1 -25238.442,E2 -25238.442} C_VEL
LIN {X 0,Y 130.664,Z 204.783,A -85,B 0,C 180,E1 -25243.633,E2 -25243.633} C_VEL
LIN {X 0,Y 131.815,Z 208.219,A -85,B 0,C 180,E1 -25244.349,E2 -25244.349} C_VEL
LIN {X 0,Y 135.374,Z 217.637,A -85,B 0,C 180,E1 -25246.48,E2 -25246.48} C_VEL
LIN {X 0,Y 136.746,Z 222.699,A -85,B 0,C 180,E1 -25247.582,E2 -25247.582} C_VEL
LIN {X 0,Y 137.739,Z 234.373,A -85,B 0,C 180,E1 -25249.941,E2 -25249.941} C_VEL
LIN {X 0,Y 138.123,Z 245.916,A -85,B 0,C 180,E1 -25252.704,E2 -25252.704} C_VEL
LIN {X 0,Y 138.05,Z 257.305,A -85,B 0,C 180,E1 -25255.945,E2 -25255.945} C_VEL
LIN {X 0,Y 137.542,Z 267.214,A -85,B 0,C 180,E1 -25259.272,E2 -25259.272} C_VEL
LIN {X 0,Y 137.234,Z 269.844,A -85,B 0,C 180,E1 -25260.25,E2 -25260.25} C_VEL
LIN {X 0,Y 133.809,Z 279.827,A -85,B 0,C 180,E1 -25264.323,E2 -25264.323} C_VEL
LIN {X 0,Y 131.041,Z 288.166,A -85,B 0,C 180,E1 -25268.776,E2 -25268.776} C_VEL
LIN {X 0,Y 128.622,Z 295.842,A -85,B 0,C 180,E1 -25274.146,E2 -25274.146} C_VEL
LIN {X 0,Y 127.46,Z 300.98,A -85,B 0,C 180,E1 -25278.873,E2 -25278.873} C_VEL
LIN {X 0,Y 127.009,Z 304.931,A -85,B 0,C 180,E1 -25283.647,E2 -25283.647} C_VEL
LIN {X 0,Y 126.994,Z 306.941,A -85,B 0,C 180,E1 -25286.828,E2 -25286.828} C_VEL
LIN {X 0,Y 127.042,Z 308.482,A -85,B 0,C 180,E1 -25290.001,E2 -25290.001} C_VEL
LIN {X 0,Y 126.8,Z 309.775,A -85,B 0,C 180,E1 -25293.893,E2 -25293.893} C_VEL
LIN {X 0,Y 126.964,Z 310.567,A -85,B 0,C 180,E1 -25299.56,E2 -25299.56} C_VEL
LIN {X 0,Y 128.439,Z 310.05,A -85,B 0,C 180,E1 -25305.879,E2 -25305.879} C_VEL
LIN {X 0,Y 131.496,Z 308.117,A -85,B 0,C 180,E1 -25311.971,E2 -25311.971} C_VEL
LIN {X 0,Y 133.597,Z 306.607,A -85,B 0,C 180,E1 -25314.889,E2 -25314.889} C_VEL
LIN {X 0,Y 138.895,Z 302.369,A -85,B 0,C 180,E1 -25320.398,E2 -25320.398} C_VEL
LIN {X 0,Y 145.288,Z 296.499,A -85,B 0,C 180,E1 -25325.485,E2 -25325.485} C_VEL
LIN {X 0,Y 152.049,Z 289.769,A -85,B 0,C 180,E1 -25329.462,E2 -25329.462} C_VEL
LIN {X 0,Y 154.94,Z 286.423,A -85,B 0,C 180,E1 -25331.127,E2 -25331.127} C_VEL
LIN {X 0,Y 159.009,Z 280.33,A -85,B 0,C 180,E1 -25334.118,E2 -25334.118} C_VEL
LIN {X 0,Y 162.549,Z 273.522,A -85,B 0,C 180,E1 -25337.309,E2 -25337.309} C_VEL
LIN {X 0,Y 164.248,Z 269.643,A -85,B 0,C 180,E1 -25339.12,E2 -25339.12} C_VEL
LIN {X 0,Y 164.9,Z 267.513,A -85,B 0,C 180,E1 -25340.259,E2 -25340.259} C_VEL
LIN {X 0,Y 165,Z 262.609,A -85,B 0,C 180,E1 -25344.027,E2 -25344.027} C_VEL
LIN {X 0,Y 164.98,Z 259.943,A -85,B 0,C 180,E1 -25346.371,E2 -25346.371} C_VEL
LIN {X 0,Y 164.881,Z 257.293,A -85,B 0,C 180,E1 -25349.235,E2 -25349.235} C_VEL
LIN {X 0,Y 164.69,Z 255.302,A -85,B 0,C 180,E1 -25352.002,E2 -25352.002} C_VEL
LIN {X 0,Y 164.547,Z 253.063,A -85,B 0,C 180,E1 -25357.392,E2 -25357.392} C_VEL
LIN {X 0,Y 164.688,Z 252.614,A -85,B 0,C 180,E1 -25360.037,E2 -25360.037} C_VEL
LIN {X 0,Y 165.434,Z 252.774,A -85,B 0,C 180,E1 -25365.231,E2 -25365.231} C_VEL
LIN {X 0,Y 165.778,Z 253.711,A -85,B 0,C 180,E1 -25367.761,E2 -25367.761} C_VEL
LIN {X 0,Y 166.098,Z 255.055,A -85,B 0,C 180,E1 -25370.255,E2 -25370.255} C_VEL
LIN {X 0,Y 166.35,Z 256.606,A -85,B 0,C 180,E1 -25372.398,E2 -25372.398} C_VEL
LIN {X 0,Y 166.153,Z 257.808,A -85,B 0,C 180,E1 -25373.446,E2 -25373.446} C_VEL
LIN {X 0,Y 164.892,Z 260.324,A -85,B 0,C 180,E1 -25374.737,E2 -25374.737} C_VEL
LIN {X 0,Y 161.42,Z 265.869,A -85,B 0,C 180,E1 -25377.187,E2 -25377.187} C_VEL
LIN {X 0,Y 160.532,Z 267.788,A -85,B 0,C 180,E1 -25378.42,E2 -25378.42} C_VEL
LIN {X 0,Y 159.439,Z 270.727,A -85,B 0,C 180,E1 -25380.63,E2 -25380.63} C_VEL
LIN {X 0,Y 158.142,Z 272.447,A -85,B 0,C 180,E1 -25381.463,E2 -25381.463} C_VEL
LIN {X 0,Y 151.245,Z 279.518,A -85,B 0,C 180,E1 -25384.691,E2 -25384.691} C_VEL
LIN {X 0,Y 144.569,Z 285.472,A -85,B 0,C 180,E1 -25388.384,E2 -25388.384} C_VEL
LIN {X 0,Y 139.613,Z 289.289,A -85,B 0,C 180,E1 -25391.615,E2 -25391.615} C_VEL
LIN {X 0,Y 135.114,Z 292.332,A -85,B 0,C 180,E1 -25395.073,E2 -25395.073} C_VEL
LIN {X 0,Y 131.167,Z 294.611,A -85,B 0,C 180,E1 -25398.751,E2 -25398.751} C_VEL
LIN {X 0,Y 127.755,Z 296.19,A -85,B 0,C 180,E1 -25402.647,E2 -25402.647} C_VEL
LIN {X 0,Y 124.878,Z 297.125,A -85,B 0,C 180,E1 -25406.757,E2 -25406.757} C_VEL
LIN {X 0,Y 122.627,Z 297.341,A -85,B 0,C 180,E1 -25411.049,E2 -25411.049} C_VEL
LIN {X 0,Y 120.936,Z 296.868,A -85,B 0,C 180,E1 -25415.551,E2 -25415.551} C_VEL
LIN {X 0,Y 119.847,Z 295.627,A -85,B 0,C 180,E1 -25420.328,E2 -25420.328} C_VEL
LIN {X 0,Y 119.406,Z 293.617,A -85,B 0,C 180,E1 -25425.065,E2 -25425.065} C_VEL
LIN {X 0,Y 119.652,Z 290.792,A -85,B 0,C 180,E1 -25429.778,E2 -25429.778} C_VEL
LIN {X 0,Y 120.534,Z 286.882,A -85,B 0,C 180,E1 -25434.713,E2 -25434.713} C_VEL
LIN {X 0,Y 121.994,Z 281.671,A -85,B 0,C 180,E1 -25439.781,E2 -25439.781} C_VEL
LIN {X 0,Y 124.211,Z 274.936,A -85,B 0,C 180,E1 -25444.859,E2 -25444.859} C_VEL
LIN {X 0,Y 127.256,Z 266.229,A -85,B 0,C 180,E1 -25449.856,E2 -25449.856} C_VEL
LIN {X 0,Y 130.505,Z 256.972,A -85,B 0,C 180,E1 -25453.978,E2 -25453.978} C_VEL
LIN {X 0,Y 133.808,Z 246.836,A -85,B 0,C 180,E1 -25457.487,E2 -25457.487} C_VEL
LIN {X 0,Y 135.119,Z 242.5,A -85,B 0,C 180,E1 -25458.752,E2 -25458.752} C_VEL
LIN {X 0,Y 134.49,Z 234.581,A -85,B 0,C 180,E1 -25461.359,E2 -25461.359} C_VEL
LIN {X 0,Y 132.956,Z 224.391,A -85,B 0,C 180,E1 -25464.444,E2 -25464.444} C_VEL
LIN {X 0,Y 130.661,Z 215.926,A -85,B 0,C 180,E1 -25466.916,E2 -25466.916} C_VEL
LIN {X 0,Y 125.737,Z 203.406,A -85,B 0,C 180,E1 -25470.629,E2 -25470.629} C_VEL
LIN {X 0,Y 124.259,Z 200.676,A -85,B 0,C 180,E1 -25471.514,E2 -25471.514} C_VEL
LIN {X 0,Y 122.847,Z 197.95,A -85,B 0,C 180,E1 -25472.377,E2 -25472.377} C_VEL
LIN {X 0,Y 122.684,Z 197.204,A -85,B 0,C 180,E1 -25472.606,E2 -25472.606} C_VEL
LIN {X 0,Y 122.454,Z 197.228,A -85,B 0,C 180,E1 -25479.914,E2 -25479.914} C_VEL
LIN {X 0,Y 122.285,Z 197.259,A -85,B 0,C 180,E1 -25483.29,E2 -25483.29} C_VEL
LIN {X 0,Y 122.071,Z 197.283,A -85,B 0,C 180,E1 -25490.208,E2 -25490.208} C_VEL
LIN {X 0,Y 121.993,Z 197.29,A -85,B 0,C 180,E1 -25493.782,E2 -25493.782} C_VEL
LIN {X 0,Y 121.923,Z 197.299,A -85,B 0,C 180,E1 -25500.162,E2 -25500.162} C_VEL
LIN {X 0,Y 121.88,Z 197.285,A -85,B 0,C 180,E1 -25506.172,E2 -25506.172} C_VEL
LIN {X 0,Y 121.869,Z 197.305,A -85,B 0,C 180,E1 -25511.439,E2 -25511.439} C_VEL
LIN {X 0,Y 121.869,Z 197.282,A -85,B 0,C 180,E1 -25518.563,E2 -25518.563} C_VEL
LIN {X 0,Y 121.931,Z 197.297,A -85,B 0,C 180,E1 -25524.805,E2 -25524.805} C_VEL
LIN {X 0,Y 121.927,Z 197.276,A -85,B 0,C 180,E1 -25529.838,E2 -25529.838} C_VEL
LIN {X 0,Y 121.995,Z 197.285,A -85,B 0,C 180,E1 -25536.22,E2 -25536.22} C_VEL
LIN {X 0,Y 122.069,Z 197.276,A -85,B 0,C 180,E1 -25539.793,E2 -25539.793} C_VEL
LIN {X 0,Y 122.241,Z 197.243,A -85,B 0,C 180,E1 -25546.706,E2 -25546.706} C_VEL
LIN {X 0,Y 122.407,Z 197.236,A -85,B 0,C 180,E1 -25550.083,E2 -25550.083} C_VEL
LIN {X 0,Y 122.599,Z 197.193,A -85,B 0,C 180,E1 -25556.715,E2 -25556.715} C_VEL
LIN {X 0,Y 123.041,Z 197.148,A -85,B 0,C 180,E1 -25560.002,E2 -25560.002} C_VEL
LIN {X 0,Y 122.419,Z 197.228,A -85,B 0,C 180,E1 -25566.595,E2 -25566.595} C_VEL
LIN {X 0,Y 122.41,Z 197.223,A -85,B 0,C 180,E1 -25569.92,E2 -25569.92} C_VEL
LIN {X 0,Y 122.247,Z 197.257,A -85,B 0,C 180,E1 -25573.296,E2 -25573.296} C_VEL
LIN {X 0,Y 122.074,Z 197.275,A -85,B 0,C 180,E1 -25580.21,E2 -25580.21} C_VEL
LIN {X 0,Y 121.999,Z 197.29,A -85,B 0,C 180,E1 -25583.783,E2 -25583.783} C_VEL
LIN {X 0,Y 122.106,Z 197.401,A -85,B 0,C 180,E1 -25587.864,E2 -25587.864} C_VEL
LIN {X 0,Y 122.29,Z 198.975,A -85,B 0,C 180,E1 -25591.148,E2 -25591.148} C_VEL
LIN {X 0,Y 122.762,Z 201.81,A -85,B 0,C 180,E1 -25596.729,E2 -25596.729} C_VEL
LIN {X 0,Y 123.364,Z 204.454,A -85,B 0,C 180,E1 -25601.479,E2 -25601.479} C_VEL
LIN {X 0,Y 124.359,Z 207.543,A -85,B 0,C 180,E1 -25602.136,E2 -25602.136} C_VEL
LIN {X 0,Y 128.129,Z 216.713,A -85,B 0,C 180,E1 -25604.488,E2 -25604.488} C_VEL
LIN {X 0,Y 130.266,Z 223.575,A -85,B 0,C 180,E1 -25606.188,E2 -25606.188} C_VEL
LIN {X 0,Y 131.204,Z 234.425,A -85,B 0,C 180,E1 -25608.585,E2 -25608.585} C_VEL
LIN {X 0,Y 131.463,Z 246.116,A -85,B 0,C 180,E1 -25611.548,E2 -25611.548} C_VEL
LIN {X 0,Y 131.238,Z 258.601,A -85,B 0,C 180,E1 -25615.321,E2 -25615.321} C_VEL
LIN {X 0,Y 130.558,Z 268.511,A -85,B 0,C 180,E1 -25618.919,E2 -25618.919} C_VEL
LIN {X 0,Y 129.253,Z 273.013,A -85,B 0,C 180,E1 -25620.702,E2 -25620.702} C_VEL
LIN {X 0,Y 125.829,Z 282.606,A -85,B 0,C 180,E1 -25625.235,E2 -25625.235} C_VEL
LIN {X 0,Y 123.147,Z 290.309,A -85,B 0,C 180,E1 -25629.976,E2 -25629.976} C_VEL
LIN {X 0,Y 121.28,Z 296.463,A -85,B 0,C 180,E1 -25634.885,E2 -25634.885} C_VEL
LIN {X 0,Y 120.223,Z 301.339,A -85,B 0,C 180,E1 -25639.9,E2 -25639.9} C_VEL
LIN {X 0,Y 119.913,Z 305.172,A -85,B 0,C 180,E1 -25645.126,E2 -25645.126} C_VEL
LIN {X 0,Y 119.982,Z 307.723,A -85,B 0,C 180,E1 -25650.001,E2 -25650.001} C_VEL
LIN {X 0,Y 119.751,Z 309.019,A -85,B 0,C 180,E1 -25653.858,E2 -25653.858} C_VEL
LIN {X 0,Y 119.948,Z 310.043,A -85,B 0,C 180,E1 -25660.124,E2 -25660.124} C_VEL
LIN {X 0,Y 121.594,Z 309.726,A -85,B 0,C 180,E1 -25666.798,E2 -25666.798} C_VEL
LIN {X 0,Y 124.918,Z 307.956,A -85,B 0,C 180,E1 -25673.193,E2 -25673.193} C_VEL
LIN {X 0,Y 129.849,Z 304.747,A -85,B 0,C 180,E1 -25679.152,E2 -25679.152} C_VEL
LIN {X 0,Y 136.048,Z 299.941,A -85,B 0,C 180,E1 -25684.628,E2 -25684.628} C_VEL
LIN {X 0,Y 141.501,Z 295.241,A -85,B 0,C 180,E1 -25688.378,E2 -25688.378} C_VEL
LIN {X 0,Y 148.754,Z 288.345,A -85,B 0,C 180,E1 -25692.319,E2 -25692.319} C_VEL
LIN {X 0,Y 153.149,Z 282.623,A -85,B 0,C 180,E1 -25695.341,E2 -25695.341} C_VEL
LIN {X 0,Y 157.054,Z 276.295,A -85,B 0,C 180,E1 -25698.578,E2 -25698.578} C_VEL
LIN {X 0,Y 159.136,Z 272.139,A -85,B 0,C 180,E1 -25700.703,E2 -25700.703} C_VEL
LIN {X 0,Y 159.65,Z 269.723,A -85,B 0,C 180,E1 -25702.41,E2 -25702.41} C_VEL
LIN {X 0,Y 159.985,Z 265.106,A -85,B 0,C 180,E1 -25706.581,E2 -25706.581} C_VEL
LIN {X 0,Y 160.131,Z 262.401,A -85,B 0,C 180,E1 -25709.686,E2 -25709.686} C_VEL
LIN {X 0,Y 160.021,Z 259.876,A -85,B 0,C 180,E1 -25713.946,E2 -25713.946} C_VEL
LIN {X 0,Y 160.042,Z 258.66,A -85,B 0,C 180,E1 -25717.249,E2 -25717.249} C_VEL
LIN {X 0,Y 160.359,Z 258.065,A -85,B 0,C 180,E1 -25722.133,E2 -25722.133} C_VEL
LIN {X 0,Y 160.811,Z 258.202,A -85,B 0,C 180,E1 -25724.797,E2 -25724.797} C_VEL
LIN {X 0,Y 161.096,Z 258.944,A -85,B 0,C 180,E1 -25727.399,E2 -25727.399} C_VEL
LIN {X 0,Y 161.283,Z 260.196,A -85,B 0,C 180,E1 -25729.961,E2 -25729.961} C_VEL
LIN {X 0,Y 161.431,Z 262.847,A -85,B 0,C 180,E1 -25733.75,E2 -25733.75} C_VEL
LIN {X 0,Y 160.864,Z 266.617,A -85,B 0,C 180,E1 -25737.495,E2 -25737.495} C_VEL
LIN {X 0,Y 160.532,Z 267.788,A -85,B 0,C 180,E1 -25738.42,E2 -25738.42} C_VEL
LIN {X 0,Y 159.565,Z 269.424,A -85,B 0,C 180,E1 -25739.329,E2 -25739.329} C_VEL
LIN {X 0,Y 156.904,Z 272.245,A -85,B 0,C 180,E1 -25740.228,E2 -25740.228} C_VEL
LIN {X 0,Y 148.828,Z 278.827,A -85,B 0,C 180,E1 -25741.814,E2 -25741.814} C_VEL
LIN {X 0,Y 147.074,Z 280.268,A -85,B 0,C 180,E1 -25742.45,E2 -25742.45} C_VEL
LIN {X 0,Y 139.343,Z 286.633,A -85,B 0,C 180,E1 -25746.515,E2 -25746.515} C_VEL
LIN {X 0,Y 132.845,Z 291.116,A -85,B 0,C 180,E1 -25750.668,E2 -25750.668} C_VEL
LIN {X 0,Y 129.801,Z 292.938,A -85,B 0,C 180,E1 -25752.938,E2 -25752.938} C_VEL
LIN {X 0,Y 125.051,Z 295.413,A -85,B 0,C 180,E1 -25757.171,E2 -25757.171} C_VEL
LIN {X 0,Y 121.009,Z 296.997,A -85,B 0,C 180,E1 -25761.679,E2 -25761.679} C_VEL
LIN {X 0,Y 117.737,Z 297.744,A -85,B 0,C 180,E1 -25766.441,E2 -25766.441} C_VEL
LIN {X 0,Y 114.395,Z 297.434,A -85,B 0,C 180,E1 -25773.566,E2 -25773.566} C_VEL
LIN {X 0,Y 113.075,Z 296.327,A -85,B 0,C 180,E1 -25778.426,E2 -25778.426} C_VEL
LIN {X 0,Y 112.383,Z 294.415,A -85,B 0,C 180,E1 -25783.461,E2 -25783.461} C_VEL
LIN {X 0,Y 112.428,Z 291.658,A -85,B 0,C 180,E1 -25788.599,E2 -25788.599} C_VEL
LIN {X 0,Y 113.468,Z 286.9,A -85,B 0,C 180,E1 -25795.02,E2 -25795.02} C_VEL
LIN {X 0,Y 115.158,Z 281.142,A -85,B 0,C 180,E1 -25800.775,E2 -25800.775} C_VEL
LIN {X 0,Y 117.646,Z 273.975,A -85,B 0,C 180,E1 -25806.219,E2 -25806.219} C_VEL
LIN {X 0,Y 120.848,Z 265.221,A -85,B 0,C 180,E1 -25811.345,E2 -25811.345} C_VEL
LIN {X 0,Y 124.228,Z 256.017,A -85,B 0,C 180,E1 -25815.476,E2 -25815.476} C_VEL
LIN {X 0,Y 127.646,Z 245.842,A -85,B 0,C 180,E1 -25819.049,E2 -25819.049} C_VEL
LIN {X 0,Y 128.5,Z 243.113,A -85,B 0,C 180,E1 -25819.877,E2 -25819.877} C_VEL
LIN {X 0,Y 127.417,Z 232.083,A -85,B 0,C 180,E1 -25823.666,E2 -25823.666} C_VEL
LIN {X 0,Y 125.853,Z 223.558,A -85,B 0,C 180,E1 -25826.397,E2 -25826.397} C_VEL
LIN {X 0,Y 123.979,Z 217.343,A -85,B 0,C 180,E1 -25828.414,E2 -25828.414} C_VEL
LIN {X 0,Y 119.559,Z 205.804,A -85,B 0,C 180,E1 -25832.18,E2 -25832.18} C_VEL
LIN {X 0,Y 116.916,Z 201.505,A -85,B 0,C 180,E1 -25833.817,E2 -25833.817} C_VEL
LIN {X 0,Y 115.58,Z 198.801,A -85,B 0,C 180,E1 -25834.741,E2 -25834.741} C_VEL
LIN {X 0,Y 115.444,Z 198.099,A -85,B 0,C 180,E1 -25835.02,E2 -25835.02} C_VEL
LIN {X 0,Y 115.369,Z 198.11,A -85,B 0,C 180,E1 -25840.53,E2 -25840.53} C_VEL
LIN {X 0,Y 115.16,Z 198.148,A -85,B 0,C 180,E1 -25844.129,E2 -25844.129} C_VEL
LIN {X 0,Y 115,Z 198.167,A -85,B 0,C 180,E1 -25851.51,E2 -25851.51} C_VEL
LIN {X 0,Y 114.872,Z 198.166,A -85,B 0,C 180,E1 -25855.357,E2 -25855.357} C_VEL
LIN {X 0,Y 114.853,Z 198.181,A -85,B 0,C 180,E1 -25861.058,E2 -25861.058} C_VEL
LIN {X 0,Y 114.776,Z 198.173,A -85,B 0,C 180,E1 -25867.757,E2 -25867.757} C_VEL
LIN {X 0,Y 114.784,Z 198.188,A -85,B 0,C 180,E1 -25872.718,E2 -25872.718} C_VEL
LIN {X 0,Y 114.792,Z 198.163,A -85,B 0,C 180,E1 -25877.668,E2 -25877.668} C_VEL
LIN {X 0,Y 114.796,Z 198.182,A -85,B 0,C 180,E1 -25882.738,E2 -25882.738} C_VEL
LIN {X 0,Y 114.86,Z 198.162,A -85,B 0,C 180,E1 -25888.939,E2 -25888.939} C_VEL
LIN {X 0,Y 114.96,Z 198.162,A -85,B 0,C 180,E1 -25896.492,E2 -25896.492} C_VEL
LIN {X 0,Y 115.026,Z 198.141,A -85,B 0,C 180,E1 -25902.214,E2 -25902.214} C_VEL
LIN {X 0,Y 115.252,Z 198.117,A -85,B 0,C 180,E1 -25907.334,E2 -25907.334} C_VEL
LIN {X 0,Y 115.366,Z 198.112,A -85,B 0,C 180,E1 -25913.004,E2 -25913.004} C_VEL
LIN {X 0,Y 115.993,Z 198.026,A -85,B 0,C 180,E1 -25920.002,E2 -25920.002} C_VEL
LIN {X 0,Y 115.361,Z 198.104,A -85,B 0,C 180,E1 -25927,E2 -25927} C_VEL
LIN {X 0,Y 115.253,Z 198.128,A -85,B 0,C 180,E1 -25932.669,E2 -25932.669} C_VEL
LIN {X 0,Y 115.033,Z 198.144,A -85,B 0,C 180,E1 -25937.789,E2 -25937.789} C_VEL
LIN {X 0,Y 114.968,Z 198.165,A -85,B 0,C 180,E1 -25943.517,E2 -25943.517} C_VEL
LIN {X 0,Y 115.037,Z 198.311,A -85,B 0,C 180,E1 -25947.273,E2 -25947.273} C_VEL
LIN {X 0,Y 115.377,Z 201.074,A -85,B 0,C 180,E1 -25953.247,E2 -25953.247} C_VEL
LIN {X 0,Y 116.008,Z 204.019,A -85,B 0,C 180,E1 -25958.976,E2 -25958.976} C_VEL
LIN {X 0,Y 117.055,Z 207.105,A -85,B 0,C 180,E1 -25959.737,E2 -25959.737} C_VEL
LIN {X 0,Y 118.179,Z 209.529,A -85,B 0,C 180,E1 -25960.461,E2 -25960.461} C_VEL
LIN {X 0,Y 121.483,Z 217.804,A -85,B 0,C 180,E1 -25962.789,E2 -25962.789} C_VEL
LIN {X 0,Y 124.012,Z 225.65,A -85,B 0,C 180,E1 -25964.962,E2 -25964.962} C_VEL
LIN {X 0,Y 124.607,Z 232.909,A -85,B 0,C 180,E1 -25966.687,E2 -25966.687} C_VEL
LIN {X 0,Y 124.893,Z 244.22,A -85,B 0,C 180,E1 -25969.675,E2 -25969.675} C_VEL
LIN {X 0,Y 124.533,Z 255.483,A -85,B 0,C 180,E1 -25973.158,E2 -25973.158} C_VEL
LIN {X 0,Y 124.025,Z 264.781,A -85,B 0,C 180,E1 -25976.56,E2 -25976.56} C_VEL
LIN {X 0,Y 123.476,Z 269.812,A -85,B 0,C 180,E1 -25978.627,E2 -25978.627} C_VEL
LIN {X 0,Y 119.933,Z 279.364,A -85,B 0,C 180,E1 -25982.991,E2 -25982.991} C_VEL
LIN {X 0,Y 116.958,Z 287.593,A -85,B 0,C 180,E1 -25987.941,E2 -25987.941} C_VEL
LIN {X 0,Y 114.996,Z 293.204,A -85,B 0,C 180,E1 -25992.208,E2 -25992.208} C_VEL
LIN {X 0,Y 113.569,Z 298.688,A -85,B 0,C 180,E1 -25997.492,E2 -25997.492} C_VEL
LIN {X 0,Y 112.917,Z 302.955,A -85,B 0,C 180,E1 -26002.85,E2 -26002.85} C_VEL
LIN {X 0,Y 112.869,Z 305.179,A -85,B 0,C 180,E1 -26006.431,E2 -26006.431} C_VEL
LIN {X 0,Y 112.922,Z 306.941,A -85,B 0,C 180,E1 -26010.001,E2 -26010.001} C_VEL
LIN {X 0,Y 112.704,Z 308.263,A -85,B 0,C 180,E1 -26013.838,E2 -26013.838} C_VEL
LIN {X 0,Y 112.957,Z 309.49,A -85,B 0,C 180,E1 -26020.758,E2 -26020.758} C_VEL
LIN {X 0,Y 114.77,Z 309.363,A -85,B 0,C 180,E1 -26027.83,E2 -26027.83} C_VEL
LIN {X 0,Y 116.326,Z 308.77,A -85,B 0,C 180,E1 -26031.254,E2 -26031.254} C_VEL
LIN {X 0,Y 120.816,Z 306.468,A -85,B 0,C 180,E1 -26037.735,E2 -26037.735} C_VEL
LIN {X 0,Y 126.81,Z 302.717,A -85,B 0,C 180,E1 -26043.658,E2 -26043.658} C_VEL
LIN {X 0,Y 132.097,Z 298.842,A -85,B 0,C 180,E1 -26047.723,E2 -26047.723} C_VEL
LIN {X 0,Y 138.132,Z 293.982,A -85,B 0,C 180,E1 -26051.409,E2 -26051.409} C_VEL
LIN {X 0,Y 143.599,Z 289.145,A -85,B 0,C 180,E1 -26054.221,E2 -26054.221} C_VEL
LIN {X 0,Y 148.182,Z 283.71,A -85,B 0,C 180,E1 -26057.32,E2 -26057.32} C_VEL
LIN {X 0,Y 152.325,Z 277.635,A -85,B 0,C 180,E1 -26060.607,E2 -26060.607} C_VEL
LIN {X 0,Y 153.919,Z 274.683,A -85,B 0,C 180,E1 -26062.405,E2 -26062.405} C_VEL
LIN {X 0,Y 154.483,Z 271.826,A -85,B 0,C 180,E1 -26064.974,E2 -26064.974} C_VEL
LIN {X 0,Y 154.919,Z 268.528,A -85,B 0,C 180,E1 -26068.553,E2 -26068.553} C_VEL
LIN {X 0,Y 155.115,Z 267.276,A -85,B 0,C 180,E1 -26070.105,E2 -26070.105} C_VEL
LIN {X 0,Y 155.181,Z 264.778,A -85,B 0,C 180,E1 -26074.93,E2 -26074.93} C_VEL
LIN {X 0,Y 155.348,Z 263.666,A -85,B 0,C 180,E1 -26078.78,E2 -26078.78} C_VEL
LIN {X 0,Y 155.928,Z 263.401,A -85,B 0,C 180,E1 -26084.309,E2 -26084.309} C_VEL
LIN {X 0,Y 156.124,Z 263.966,A -85,B 0,C 180,E1 -26086.991,E2 -26086.991} C_VEL
LIN {X 0,Y 156.246,Z 265.085,A -85,B 0,C 180,E1 -26089.633,E2 -26089.633} C_VEL
LIN {X 0,Y 156.071,Z 267.594,A -85,B 0,C 180,E1 -26093.535,E2 -26093.535} C_VEL
LIN {X 0,Y 155.535,Z 269.914,A -85,B 0,C 180,E1 -26096.112,E2 -26096.112} C_VEL
LIN {X 0,Y 154.412,Z 272.662,A -85,B 0,C 180,E1 -26098.564,E2 -26098.564} C_VEL
LIN {X 0,Y 153.97,Z 273.532,A -85,B 0,C 180,E1 -26099.279,E2 -26099.279} C_VEL
LIN {X 0,Y 147.074,Z 280.268,A -85,B 0,C 180,E1 -26102.45,E2 -26102.45} C_VEL
LIN {X 0,Y 143.357,Z 283.204,A -85,B 0,C 180,E1 -26103.858,E2 -26103.858} C_VEL
LIN {X 0,Y 136.048,Z 287.718,A -85,B 0,C 180,E1 -26105.903,E2 -26105.903} C_VEL
LIN {X 0,Y 128.767,Z 291.509,A -85,B 0,C 180,E1 -26108.29,E2 -26108.29} C_VEL
LIN {X 0,Y 125.196,Z 293.268,A -85,B 0,C 180,E1 -26110.248,E2 -26110.248} C_VEL
LIN {X 0,Y 121.242,Z 295.225,A -85,B 0,C 180,E1 -26113.405,E2 -26113.405} C_VEL
LIN {X 0,Y 116.997,Z 296.942,A -85,B 0,C 180,E1 -26117.477,E2 -26117.477} C_VEL
LIN {X 0,Y 113.34,Z 297.958,A -85,B 0,C 180,E1 -26121.84,E2 -26121.84} C_VEL
LIN {X 0,Y 110.207,Z 298.294,A -85,B 0,C 180,E1 -26126.772,E2 -26126.772} C_VEL
LIN {X 0,Y 107.758,Z 297.881,A -85,B 0,C 180,E1 -26132.019,E2 -26132.019} C_VEL
LIN {X 0,Y 106.161,Z 296.693,A -85,B 0,C 180,E1 -26137.398,E2 -26137.398} C_VEL
LIN {X 0,Y 105.232,Z 293.593,A -85,B 0,C 180,E1 -26145.159,E2 -26145.159} C_VEL
LIN {X 0,Y 105.889,Z 288.914,A -85,B 0,C 180,E1 -26152.79,E2 -26152.79} C_VEL
LIN {X 0,Y 107.212,Z 284.136,A -85,B 0,C 180,E1 -26158.446,E2 -26158.446} C_VEL
LIN {X 0,Y 109.326,Z 277.857,A -85,B 0,C 180,E1 -26164.152,E2 -26164.152} C_VEL
LIN {X 0,Y 112.318,Z 269.769,A -85,B 0,C 180,E1 -26169.81,E2 -26169.81} C_VEL
LIN {X 0,Y 115.838,Z 260.826,A -85,B 0,C 180,E1 -26174.58,E2 -26174.58} C_VEL
LIN {X 0,Y 119.787,Z 249.966,A -85,B 0,C 180,E1 -26179.007,E2 -26179.007} C_VEL
LIN {X 0,Y 121.679,Z 244.393,A -85,B 0,C 180,E1 -26180.86,E2 -26180.86} C_VEL
LIN {X 0,Y 121.119,Z 235.446,A -85,B 0,C 180,E1 -26184.171,E2 -26184.171} C_VEL
LIN {X 0,Y 119.755,Z 226.676,A -85,B 0,C 180,E1 -26187.232,E2 -26187.232} C_VEL
LIN {X 0,Y 118.056,Z 220.668,A -85,B 0,C 180,E1 -26189.394,E2 -26189.394} C_VEL
LIN {X 0,Y 114.601,Z 210.957,A -85,B 0,C 180,E1 -26192.818,E2 -26192.818} C_VEL
LIN {X 0,Y 110.413,Z 203.285,A -85,B 0,C 180,E1 -26195.935,E2 -26195.935} C_VEL
LIN {X 0,Y 108.609,Z 200.221,A -85,B 0,C 180,E1 -26197.26,E2 -26197.26} C_VEL
LIN {X 0,Y 108.319,Z 198.997,A -85,B 0,C 180,E1 -26197.69,E2 -26197.69} C_VEL
LIN {X 0,Y 108.213,Z 199.012,A -85,B 0,C 180,E1 -26203.055,E2 -26203.055} C_VEL
LIN {X 0,Y 107.923,Z 199.039,A -85,B 0,C 180,E1 -26209.002,E2 -26209.002} C_VEL
LIN {X 0,Y 107.865,Z 199.047,A -85,B 0,C 180,E1 -26214.197,E2 -26214.197} C_VEL
LIN {X 0,Y 107.776,Z 199.061,A -85,B 0,C 180,E1 -26222.039,E2 -26222.039} C_VEL
LIN {X 0,Y 107.685,Z 199.06,A -85,B 0,C 180,E1 -26228.451,E2 -26228.451} C_VEL
LIN {X 0,Y 107.674,Z 199.059,A -85,B 0,C 180,E1 -26235.887,E2 -26235.887} C_VEL
LIN {X 0,Y 107.692,Z 199.062,A -85,B 0,C 180,E1 -26241.546,E2 -26241.546} C_VEL
LIN {X 0,Y 107.798,Z 199.042,A -85,B 0,C 180,E1 -26248.565,E2 -26248.565} C_VEL
LIN {X 0,Y 107.925,Z 199.04,A -85,B 0,C 180,E1 -26257.003,E2 -26257.003} C_VEL
LIN {X 0,Y 108.035,Z 199.002,A -85,B 0,C 180,E1 -26264.919,E2 -26264.919} C_VEL
LIN {X 0,Y 108.253,Z 198.995,A -85,B 0,C 180,E1 -26268.771,E2 -26268.771} C_VEL
LIN {X 0,Y 108.447,Z 198.956,A -85,B 0,C 180,E1 -26276.286,E2 -26276.286} C_VEL
LIN {X 0,Y 108.918,Z 198.907,A -85,B 0,C 180,E1 -26280.002,E2 -26280.002} C_VEL
LIN {X 0,Y 108.301,Z 198.98,A -85,B 0,C 180,E1 -26287.459,E2 -26287.459} C_VEL
LIN {X 0,Y 108.174,Z 199.01,A -85,B 0,C 180,E1 -26292.958,E2 -26292.958} C_VEL
LIN {X 0,Y 107.928,Z 199.03,A -85,B 0,C 180,E1 -26299.003,E2 -26299.003} C_VEL
LIN {X 0,Y 107.928,Z 199.043,A -85,B 0,C 180,E1 -26305.879,E2 -26305.879} C_VEL
LIN {X 0,Y 108.302,Z 201.701,A -85,B 0,C 180,E1 -26312.479,E2 -26312.479} C_VEL
LIN {X 0,Y 108.583,Z 203.391,A -85,B 0,C 180,E1 -26316.057,E2 -26316.057} C_VEL
LIN {X 0,Y 109.658,Z 206.554,A -85,B 0,C 180,E1 -26316.924,E2 -26316.924} C_VEL
LIN {X 0,Y 110.866,Z 208.792,A -85,B 0,C 180,E1 -26317.73,E2 -26317.73} C_VEL
LIN {X 0,Y 114.575,Z 218.082,A -85,B 0,C 180,E1 -26320.675,E2 -26320.675} C_VEL
LIN {X 0,Y 117.515,Z 227.05,A -85,B 0,C 180,E1 -26323.458,E2 -26323.458} C_VEL
LIN {X 0,Y 118.156,Z 231.534,A -85,B 0,C 180,E1 -26324.691,E2 -26324.691} C_VEL
LIN {X 0,Y 118.316,Z 242.855,A -85,B 0,C 180,E1 -26327.777,E2 -26327.777} C_VEL
LIN {X 0,Y 117.959,Z 253.797,A -85,B 0,C 180,E1 -26331.275,E2 -26331.275} C_VEL
LIN {X 0,Y 117.24,Z 264.258,A -85,B 0,C 180,E1 -26335.286,E2 -26335.286} C_VEL
LIN {X 0,Y 116.489,Z 270.239,A -85,B 0,C 180,E1 -26337.9,E2 -26337.9} C_VEL
LIN {X 0,Y 113.028,Z 279.07,A -85,B 0,C 180,E1 -26342.203,E2 -26342.203} C_VEL
LIN {X 0,Y 109.914,Z 287.264,A -85,B 0,C 180,E1 -26347.441,E2 -26347.441} C_VEL
LIN {X 0,Y 107.582,Z 293.847,A -85,B 0,C 180,E1 -26352.905,E2 -26352.905} C_VEL
LIN {X 0,Y 106.276,Z 299.093,A -85,B 0,C 180,E1 -26358.558,E2 -26358.558} C_VEL
LIN {X 0,Y 105.804,Z 303.673,A -85,B 0,C 180,E1 -26365.139,E2 -26365.139} C_VEL
LIN {X 0,Y 105.862,Z 306.079,A -85,B 0,C 180,E1 -26370.001,E2 -26370.001} C_VEL
LIN {X 0,Y 105.657,Z 307.435,A -85,B 0,C 180,E1 -26373.815,E2 -26373.815} C_VEL
LIN {X 0,Y 105.964,Z 308.933,A -85,B 0,C 180,E1 -26381.478,E2 -26381.478} C_VEL
LIN {X 0,Y 107.992,Z 308.965,A -85,B 0,C 180,E1 -26388.99,E2 -26388.99} C_VEL
LIN {X 0,Y 111.974,Z 307.621,A -85,B 0,C 180,E1 -26396.063,E2 -26396.063} C_VEL
LIN {X 0,Y 114.563,Z 306.418,A -85,B 0,C 180,E1 -26399.392,E2 -26399.392} C_VEL
LIN {X 0,Y 121.125,Z 302.743,A -85,B 0,C 180,E1 -26405.674,E2 -26405.674} C_VEL
LIN {X 0,Y 128.587,Z 297.783,A -85,B 0,C 180,E1 -26410.986,E2 -26410.986} C_VEL
LIN {X 0,Y 135.221,Z 292.81,A -85,B 0,C 180,E1 -26414.56,E2 -26414.56} C_VEL
LIN {X 0,Y 137.528,Z 290.904,A -85,B 0,C 180,E1 -26415.68,E2 -26415.68} C_VEL
LIN {X 0,Y 142.463,Z 285.846,A -85,B 0,C 180,E1 -26418.769,E2 -26418.769} C_VEL
LIN {X 0,Y 146.964,Z 280.21,A -85,B 0,C 180,E1 -26422.095,E2 -26422.095} C_VEL
LIN {X 0,Y 148.394,Z 277.925,A -85,B 0,C 180,E1 -26423.624,E2 -26423.624} C_VEL
LIN {X 0,Y 149.302,Z 274.498,A -85,B 0,C 180,E1 -26427.226,E2 -26427.226} C_VEL
LIN {X 0,Y 149.846,Z 271.94,A -85,B 0,C 180,E1 -26430.496,E2 -26430.496} C_VEL
LIN {X 0,Y 150.083,Z 269.738,A -85,B 0,C 180,E1 -26435.073,E2 -26435.073} C_VEL
LIN {X 0,Y 150.338,Z 268.639,A -85,B 0,C 180,E1 -26439.224,E2 -26439.224} C_VEL
LIN {X 0,Y 150.742,Z 268.362,A -85,B 0,C 180,E1 -26443.754,E2 -26443.754} C_VEL
LIN {X 0,Y 150.946,Z 268.763,A -85,B 0,C 180,E1 -26446.537,E2 -26446.537} C_VEL
LIN {X 0,Y 150.97,Z 269.743,A -85,B 0,C 180,E1 -26449.267,E2 -26449.267} C_VEL
LIN {X 0,Y 150.731,Z 271.179,A -85,B 0,C 180,E1 -26451.958,E2 -26451.958} C_VEL
LIN {X 0,Y 150.156,Z 273.163,A -85,B 0,C 180,E1 -26454.627,E2 -26454.627} C_VEL
LIN {X 0,Y 148.906,Z 275.708,A -85,B 0,C 180,E1 -26457.293,E2 -26457.293} C_VEL
LIN {X 0,Y 147.545,Z 277.17,A -85,B 0,C 180,E1 -26458.191,E2 -26458.191} C_VEL
LIN {X 0,Y 139.161,Z 284.24,A -85,B 0,C 180,E1 -26461.944,E2 -26461.944} C_VEL
LIN {X 0,Y 131.431,Z 289.676,A -85,B 0,C 180,E1 -26466.138,E2 -26466.138} C_VEL
LIN {X 0,Y 125.196,Z 293.268,A -85,B 0,C 180,E1 -26470.248,E2 -26470.248} C_VEL
LIN {X 0,Y 121.718,Z 294.85,A -85,B 0,C 180,E1 -26472.361,E2 -26472.361} C_VEL
LIN {X 0,Y 114.827,Z 297.016,A -85,B 0,C 180,E1 -26475.665,E2 -26475.665} C_VEL
LIN {X 0,Y 108.309,Z 298.381,A -85,B 0,C 180,E1 -26479.424,E2 -26479.424} C_VEL
LIN {X 0,Y 105.541,Z 298.708,A -85,B 0,C 180,E1 -26482.206,E2 -26482.206} C_VEL
LIN {X 0,Y 101.78,Z 298.518,A -85,B 0,C 180,E1 -26488.903,E2 -26488.903} C_VEL
LIN {X 0,Y 99.794,Z 297.525,A -85,B 0,C 180,E1 -26494.289,E2 -26494.289} C_VEL
LIN {X 0,Y 98.554,Z 295.816,A -85,B 0,C 180,E1 -26499.923,E2 -26499.923} C_VEL
LIN {X 0,Y 98.209,Z 292.132,A -85,B 0,C 180,E1 -26507.869,E2 -26507.869} C_VEL
LIN {X 0,Y 98.901,Z 288.44,A -85,B 0,C 180,E1 -26513.6,E2 -26513.6} C_VEL
LIN {X 0,Y 100.754,Z 282.351,A -85,B 0,C 180,E1 -26520.772,E2 -26520.772} C_VEL
LIN {X 0,Y 103.278,Z 275.45,A -85,B 0,C 180,E1 -26526.854,E2 -26526.854} C_VEL
LIN {X 0,Y 106.819,Z 266.61,A -85,B 0,C 180,E1 -26532.777,E2 -26532.777} C_VEL
LIN {X 0,Y 110.657,Z 257.031,A -85,B 0,C 180,E1 -26537.622,E2 -26537.622} C_VEL
LIN {X 0,Y 114.916,Z 245.561,A -85,B 0,C 180,E1 -26541.98,E2 -26541.98} C_VEL
LIN {X 0,Y 114.968,Z 241.933,A -85,B 0,C 180,E1 -26543.418,E2 -26543.418} C_VEL
LIN {X 0,Y 114.14,Z 232.914,A -85,B 0,C 180,E1 -26546.911,E2 -26546.911} C_VEL
LIN {X 0,Y 112.444,Z 225.018,A -85,B 0,C 180,E1 -26549.929,E2 -26549.929} C_VEL
LIN {X 0,Y 109.245,Z 215.489,A -85,B 0,C 180,E1 -26553.688,E2 -26553.688} C_VEL
LIN {X 0,Y 104.539,Z 206.626,A -85,B 0,C 180,E1 -26557.727,E2 -26557.727} C_VEL
LIN {X 0,Y 102.953,Z 203.622,A -85,B 0,C 180,E1 -26559.066,E2 -26559.066} C_VEL
LIN {X 0,Y 101.448,Z 200.881,A -85,B 0,C 180,E1 -26560.351,E2 -26560.351} C_VEL
LIN {X 0,Y 101.258,Z 199.867,A -85,B 0,C 180,E1 -26560.75,E2 -26560.75} C_VEL
LIN {X 0,Y 100.937,Z 199.912,A -85,B 0,C 180,E1 -26566.171,E2 -26566.171} C_VEL
LIN {X 0,Y 100.831,Z 199.93,A -85,B 0,C 180,E1 -26570.395,E2 -26570.395} C_VEL
LIN {X 0,Y 100.771,Z 199.924,A -85,B 0,C 180,E1 -26574.959,E2 -26574.959} C_VEL
LIN {X 0,Y 100.685,Z 199.94,A -85,B 0,C 180,E1 -26583.114,E2 -26583.114} C_VEL
LIN {X 0,Y 100.637,Z 199.944,A -85,B 0,C 180,E1 -26589.812,E2 -26589.812} C_VEL
LIN {X 0,Y 100.645,Z 199.934,A -85,B 0,C 180,E1 -26595.712,E2 -26595.712} C_VEL
LIN {X 0,Y 100.63,Z 199.939,A -85,B 0,C 180,E1 -26601.059,E2 -26601.059} C_VEL
LIN {X 0,Y 100.692,Z 199.936,A -85,B 0,C 180,E1 -26606.882,E2 -26606.882} C_VEL
LIN {X 0,Y 100.784,Z 199.924,A -85,B 0,C 180,E1 -26615.269,E2 -26615.269} C_VEL
LIN {X 0,Y 100.83,Z 199.922,A -85,B 0,C 180,E1 -26619.606,E2 -26619.606} C_VEL
LIN {X 0,Y 101.101,Z 199.873,A -85,B 0,C 180,E1 -26626.703,E2 -26626.703} C_VEL
LIN {X 0,Y 101.243,Z 199.873,A -85,B 0,C 180,E1 -26632.022,E2 -26632.022} C_VEL
LIN {X 0,Y 101.846,Z 199.787,A -85,B 0,C 180,E1 -26640.002,E2 -26640.002} C_VEL
LIN {X 0,Y 101.241,Z 199.856,A -85,B 0,C 180,E1 -26647.983,E2 -26647.983} C_VEL
LIN {X 0,Y 101.103,Z 199.891,A -85,B 0,C 180,E1 -26653.301,E2 -26653.301} C_VEL
LIN {X 0,Y 100.838,Z 199.92,A -85,B 0,C 180,E1 -26660.397,E2 -26660.397} C_VEL
LIN {X 0,Y 100.904,Z 200.014,A -85,B 0,C 180,E1 -26665.696,E2 -26665.696} C_VEL
LIN {X 0,Y 101.292,Z 202.861,A -85,B 0,C 180,E1 -26672.718,E2 -26672.718} C_VEL
LIN {X 0,Y 102.272,Z 205.992,A -85,B 0,C 180,E1 -26673.676,E2 -26673.676} C_VEL
LIN {X 0,Y 103.689,Z 208.637,A -85,B 0,C 180,E1 -26674.78,E2 -26674.78} C_VEL
LIN {X 0,Y 106.693,Z 215.599,A -85,B 0,C 180,E1 -26677.329,E2 -26677.329} C_VEL
LIN {X 0,Y 110.044,Z 224.919,A -85,B 0,C 180,E1 -26680.592,E2 -26680.592} C_VEL
LIN {X 0,Y 111.656,Z 230.76,A -85,B 0,C 180,E1 -26682.584,E2 -26682.584} C_VEL
LIN {X 0,Y 111.868,Z 241.094,A -85,B 0,C 180,E1 -26685.606,E2 -26685.606} C_VEL
LIN {X 0,Y 111.437,Z 251.875,A -85,B 0,C 180,E1 -26689.186,E2 -26689.186} C_VEL
LIN {X 0,Y 110.635,Z 262.69,A -85,B 0,C 180,E1 -26693.449,E2 -26693.449} C_VEL
LIN {X 0,Y 109.86,Z 269.405,A -85,B 0,C 180,E1 -26696.539,E2 -26696.539} C_VEL
LIN {X 0,Y 106.154,Z 278.691,A -85,B 0,C 180,E1 -26701.316,E2 -26701.316} C_VEL
LIN {X 0,Y 102.887,Z 286.849,A -85,B 0,C 180,E1 -26706.874,E2 -26706.874} C_VEL
LIN {X 0,Y 100.815,Z 292.421,A -85,B 0,C 180,E1 -26711.718,E2 -26711.718} C_VEL
LIN {X 0,Y 99.344,Z 297.865,A -85,B 0,C 180,E1 -26717.747,E2 -26717.747} C_VEL
LIN {X 0,Y 98.771,Z 302.755,A -85,B 0,C 180,E1 -26725.001,E2 -26725.001} C_VEL
LIN {X 0,Y 98.804,Z 305.207,A -85,B 0,C 180,E1 -26730.001,E2 -26730.001} C_VEL
LIN {X 0,Y 98.603,Z 306.643,A -85,B 0,C 180,E1 -26734.088,E2 -26734.088} C_VEL
LIN {X 0,Y 99.004,Z 308.334,A -85,B 0,C 180,E1 -26742.297,E2 -26742.297} C_VEL
LIN {X 0,Y 101.269,Z 308.57,A -85,B 0,C 180,E1 -26750.305,E2 -26750.305} C_VEL
LIN {X 0,Y 105.616,Z 307.4,A -85,B 0,C 180,E1 -26757.763,E2 -26757.763} C_VEL
LIN {X 0,Y 111.682,Z 304.848,A -85,B 0,C 180,E1 -26764.498,E2 -26764.498} C_VEL
LIN {X 0,Y 119.119,Z 300.8,A -85,B 0,C 180,E1 -26770.467,E2 -26770.467} C_VEL
LIN {X 0,Y 125.571,Z 296.725,A -85,B 0,C 180,E1 -26774.396,E2 -26774.396} C_VEL
LIN {X 0,Y 132.674,Z 291.651,A -85,B 0,C 180,E1 -26777.87,E2 -26777.87} C_VEL
LIN {X 0,Y 136.861,Z 287.818,A -85,B 0,C 180,E1 -26780.379,E2 -26780.379} C_VEL
LIN {X 0,Y 141.124,Z 283.234,A -85,B 0,C 180,E1 -26783.3,E2 -26783.3} C_VEL
LIN {X 0,Y 142.513,Z 281.519,A -85,B 0,C 180,E1 -26784.457,E2 -26784.457} C_VEL
LIN {X 0,Y 143.543,Z 278.883,A -85,B 0,C 180,E1 -26787.412,E2 -26787.412} C_VEL
LIN {X 0,Y 144.376,Z 276.18,A -85,B 0,C 180,E1 -26791.19,E2 -26791.19} C_VEL
LIN {X 0,Y 144.606,Z 274.865,A -85,B 0,C 180,E1 -26794.06,E2 -26794.06} C_VEL
LIN {X 0,Y 144.803,Z 273.824,A -85,B 0,C 180,E1 -26797.246,E2 -26797.246} C_VEL
LIN {X 0,Y 145.085,Z 273.242,A -85,B 0,C 180,E1 -26800.177,E2 -26800.177} C_VEL
LIN {X 0,Y 145.46,Z 273.208,A -85,B 0,C 180,E1 -26805.089,E2 -26805.089} C_VEL
LIN {X 0,Y 145.482,Z 274.142,A -85,B 0,C 180,E1 -26808.857,E2 -26808.857} C_VEL
LIN {X 0,Y 145.067,Z 275.47,A -85,B 0,C 180,E1 -26811.642,E2 -26811.642} C_VEL
LIN {X 0,Y 144.198,Z 277.338,A -85,B 0,C 180,E1 -26814.405,E2 -26814.405} C_VEL
LIN {X 0,Y 143.496,Z 278.476,A -85,B 0,C 180,E1 -26815.751,E2 -26815.751} C_VEL
LIN {X 0,Y 142.361,Z 279.569,A -85,B 0,C 180,E1 -26816.409,E2 -26816.409} C_VEL
LIN {X 0,Y 133.535,Z 286.221,A -85,B 0,C 180,E1 -26820.224,E2 -26820.224} C_VEL
LIN {X 0,Y 124.624,Z 291.771,A -85,B 0,C 180,E1 -26825.012,E2 -26825.012} C_VEL
LIN {X 0,Y 116.74,Z 295.575,A -85,B 0,C 180,E1 -26830.403,E2 -26830.403} C_VEL
LIN {X 0,Y 110.016,Z 297.908,A -85,B 0,C 180,E1 -26836.616,E2 -26836.616} C_VEL
LIN {X 0,Y 105.541,Z 298.708,A -85,B 0,C 180,E1 -26842.206,E2 -26842.206} C_VEL
LIN {X 0,Y 103.005,Z 298.817,A -85,B 0,C 180,E1 -26845.142,E2 -26845.142} C_VEL
LIN {X 0,Y 97.693,Z 298.437,A -85,B 0,C 180,E1 -26849.928,E2 -26849.928} C_VEL
LIN {X 0,Y 93.792,Z 297.596,A -85,B 0,C 180,E1 -26854.06,E2 -26854.06} C_VEL
LIN {X 0,Y 91.918,Z 296.583,A -85,B 0,C 180,E1 -26857.478,E2 -26857.478} C_VEL
LIN {X 0,Y 91.617,Z 296.155,A -85,B 0,C 180,E1 -26858.672,E2 -26858.672} C_VEL
LIN {X 0,Y 91.045,Z 293.058,A -85,B 0,C 180,E1 -26865.993,E2 -26865.993} C_VEL
LIN {X 0,Y 91.963,Z 287.901,A -85,B 0,C 180,E1 -26874.62,E2 -26874.62} C_VEL
LIN {X 0,Y 94.014,Z 281.583,A -85,B 0,C 180,E1 -26882.148,E2 -26882.148} C_VEL
LIN {X 0,Y 96.862,Z 274.26,A -85,B 0,C 180,E1 -26888.728,E2 -26888.728} C_VEL
LIN {X 0,Y 100.266,Z 266.182,A -85,B 0,C 180,E1 -26894.273,E2 -26894.273} C_VEL
LIN {X 0,Y 104.199,Z 256.784,A -85,B 0,C 180,E1 -26899.173,E2 -26899.173} C_VEL
LIN {X 0,Y 108.426,Z 245.999,A -85,B 0,C 180,E1 -26903.449,E2 -26903.449} C_VEL
LIN {X 0,Y 107.987,Z 237.192,A -85,B 0,C 180,E1 -26907.202,E2 -26907.202} C_VEL
LIN {X 0,Y 106.989,Z 230.446,A -85,B 0,C 180,E1 -26909.999,E2 -26909.999} C_VEL
LIN {X 0,Y 103.581,Z 219.103,A -85,B 0,C 180,E1 -26914.926,E2 -26914.926} C_VEL
LIN {X 0,Y 98.701,Z 209.487,A -85,B 0,C 180,E1 -26919.733,E2 -26919.733} C_VEL
LIN {X 0,Y 96.127,Z 204.828,A -85,B 0,C 180,E1 -26922.23,E2 -26922.23} C_VEL
LIN {X 0,Y 94.33,Z 202.097,A -85,B 0,C 180,E1 -26923.905,E2 -26923.905} C_VEL
LIN {X 0,Y 93.979,Z 200.787,A -85,B 0,C 180,E1 -26924.529,E2 -26924.529} C_VEL
LIN {X 0,Y 93.701,Z 200.82,A -85,B 0,C 180,E1 -26932.025,E2 -26932.025} C_VEL
LIN {X 0,Y 93.617,Z 200.81,A -85,B 0,C 180,E1 -26936.771,E2 -26936.771} C_VEL
LIN {X 0,Y 93.582,Z 200.816,A -85,B 0,C 180,E1 -26944.304,E2 -26944.304} C_VEL
LIN {X 0,Y 93.53,Z 200.835,A -85,B 0,C 180,E1 -26952.553,E2 -26952.553} C_VEL
LIN {X 0,Y 93.535,Z 200.809,A -85,B 0,C 180,E1 -26958.709,E2 -26958.709} C_VEL
LIN {X 0,Y 93.59,Z 200.825,A -85,B 0,C 180,E1 -26965.692,E2 -26965.692} C_VEL
LIN {X 0,Y 93.667,Z 200.804,A -85,B 0,C 180,E1 -26974.207,E2 -26974.207} C_VEL
LIN {X 0,Y 93.701,Z 200.812,A -85,B 0,C 180,E1 -26977.977,E2 -26977.977} C_VEL
LIN {X 0,Y 94.021,Z 200.752,A -85,B 0,C 180,E1 -26986.343,E2 -26986.343} C_VEL
LIN {X 0,Y 94.176,Z 200.754,A -85,B 0,C 180,E1 -26991.419,E2 -26991.419} C_VEL
LIN {X 0,Y 94.774,Z 200.667,A -85,B 0,C 180,E1 -27000.002,E2 -27000.002} C_VEL
LIN {X 0,Y 94.174,Z 200.735,A -85,B 0,C 180,E1 -27008.586,E2 -27008.586} C_VEL
LIN {X 0,Y 94.023,Z 200.774,A -85,B 0,C 180,E1 -27013.661,E2 -27013.661} C_VEL
LIN {X 0,Y 93.735,Z 200.809,A -85,B 0,C 180,E1 -27022.02,E2 -27022.02} C_VEL
LIN {X 0,Y 93.821,Z 200.842,A -85,B 0,C 180,E1 -27024.822,E2 -27024.822} C_VEL
LIN {X 0,Y 94.034,Z 202.291,A -85,B 0,C 180,E1 -27028.762,E2 -27028.762} C_VEL
LIN {X 0,Y 95.204,Z 205.705,A -85,B 0,C 180,E1 -27030.042,E2 -27030.042} C_VEL
LIN {X 0,Y 96.532,Z 208.027,A -85,B 0,C 180,E1 -27031.194,E2 -27031.194} C_VEL
LIN {X 0,Y 98.282,Z 211.973,A -85,B 0,C 180,E1 -27032.876,E2 -27032.876} C_VEL
LIN {X 0,Y 101.6,Z 220.394,A -85,B 0,C 180,E1 -27036.322,E2 -27036.322} C_VEL
LIN {X 0,Y 104.925,Z 230.882,A -85,B 0,C 180,E1 -27040.374,E2 -27040.374} C_VEL
LIN {X 0,Y 105.612,Z 234.677,A -85,B 0,C 180,E1 -27041.72,E2 -27041.72} C_VEL
LIN {X 0,Y 105.278,Z 246.259,A -85,B 0,C 180,E1 -27045.501,E2 -27045.501} C_VEL
LIN {X 0,Y 104.422,Z 257.024,A -85,B 0,C 180,E1 -27049.625,E2 -27049.625} C_VEL
LIN {X 0,Y 103.464,Z 266.487,A -85,B 0,C 180,E1 -27053.961,E2 -27053.961} C_VEL
LIN {X 0,Y 102.834,Z 269.996,A -85,B 0,C 180,E1 -27055.74,E2 -27055.74} C_VEL
LIN {X 0,Y 99.32,Z 278.264,A -85,B 0,C 180,E1 -27060.309,E2 -27060.309} C_VEL
LIN {X 0,Y 95.897,Z 286.417,A -85,B 0,C 180,E1 -27066.23,E2 -27066.23} C_VEL
LIN {X 0,Y 93.41,Z 292.972,A -85,B 0,C 180,E1 -27072.486,E2 -27072.486} C_VEL
LIN {X 0,Y 92.058,Z 298.204,A -85,B 0,C 180,E1 -27078.998,E2 -27078.998} C_VEL
LIN {X 0,Y 91.726,Z 302.243,A -85,B 0,C 180,E1 -27085.606,E2 -27085.606} C_VEL
LIN {X 0,Y 91.746,Z 304.308,A -85,B 0,C 180,E1 -27090.001,E2 -27090.001} C_VEL
LIN {X 0,Y 91.541,Z 305.83,A -85,B 0,C 180,E1 -27094.404,E2 -27094.404} C_VEL
LIN {X 0,Y 92.078,Z 307.681,A -85,B 0,C 180,E1 -27103.238,E2 -27103.238} C_VEL
LIN {X 0,Y 94.611,Z 308.131,A -85,B 0,C 180,E1 -27111.804,E2 -27111.804} C_VEL
LIN {X 0,Y 99.354,Z 307.192,A -85,B 0,C 180,E1 -27119.681,E2 -27119.681} C_VEL
LIN {X 0,Y 105.879,Z 304.836,A -85,B 0,C 180,E1 -27126.685,E2 -27126.685} C_VEL
LIN {X 0,Y 113.82,Z 301.05,A -85,B 0,C 180,E1 -27132.783,E2 -27132.783} C_VEL
LIN {X 0,Y 120.619,Z 297.186,A -85,B 0,C 180,E1 -27136.747,E2 -27136.747} C_VEL
LIN {X 0,Y 128.013,Z 292.363,A -85,B 0,C 180,E1 -27140.23,E2 -27140.23} C_VEL
LIN {X 0,Y 132.372,Z 288.739,A -85,B 0,C 180,E1 -27142.788,E2 -27142.788} C_VEL
LIN {X 0,Y 136.441,Z 284.842,A -85,B 0,C 180,E1 -27145.504,E2 -27145.504} C_VEL
LIN {X 0,Y 137.568,Z 282.978,A -85,B 0,C 180,E1 -27147.567,E2 -27147.567} C_VEL
LIN {X 0,Y 138.237,Z 281.431,A -85,B 0,C 180,E1 -27149.802,E2 -27149.802} C_VEL
LIN {X 0,Y 138.822,Z 279.77,A -85,B 0,C 180,E1 -27152.893,E2 -27152.893} C_VEL
LIN {X 0,Y 139.089,Z 278.594,A -85,B 0,C 180,E1 -27156.156,E2 -27156.156} C_VEL
LIN {X 0,Y 139.421,Z 277.844,A -85,B 0,C 180,E1 -27159.336,E2 -27159.336} C_VEL
LIN {X 0,Y 139.705,Z 277.506,A -85,B 0,C 180,E1 -27162.906,E2 -27162.906} C_VEL
LIN {X 0,Y 139.888,Z 277.637,A -85,B 0,C 180,E1 -27165.45,E2 -27165.45} C_VEL
LIN {X 0,Y 139.766,Z 278.267,A -85,B 0,C 180,E1 -27168.395,E2 -27168.395} C_VEL
LIN {X 0,Y 139.206,Z 279.493,A -85,B 0,C 180,E1 -27171.287,E2 -27171.287} C_VEL
LIN {X 0,Y 138.015,Z 281.255,A -85,B 0,C 180,E1 -27174.153,E2 -27174.153} C_VEL
LIN {X 0,Y 128.871,Z 287.648,A -85,B 0,C 180,E1 -27177.977,E2 -27177.977} C_VEL
LIN {X 0,Y 122.069,Z 291.573,A -85,B 0,C 180,E1 -27181.325,E2 -27181.325} C_VEL
LIN {X 0,Y 113.229,Z 295.693,A -85,B 0,C 180,E1 -27186.725,E2 -27186.725} C_VEL
LIN {X 0,Y 107.447,Z 297.722,A -85,B 0,C 180,E1 -27191.314,E2 -27191.314} C_VEL
LIN {X 0,Y 102.487,Z 298.875,A -85,B 0,C 180,E1 -27196.248,E2 -27196.248} C_VEL
LIN {X 0,Y 98.326,Z 299.259,A -85,B 0,C 180,E1 -27201.688,E2 -27201.688} C_VEL
LIN {X 0,Y 95.082,Z 298.876,A -85,B 0,C 180,E1 -27207.502,E2 -27207.502} C_VEL
LIN {X 0,Y 92.797,Z 297.708,A -85,B 0,C 180,E1 -27213.581,E2 -27213.581} C_VEL
LIN {X 0,Y 91.617,Z 296.155,A -85,B 0,C 180,E1 -27218.672,E2 -27218.672} C_VEL
LIN {X 0,Y 90.512,Z 294.794,A -85,B 0,C 180,E1 -27222.209,E2 -27222.209} C_VEL
LIN {X 0,Y 87.574,Z 291.976,A -85,B 0,C 180,E1 -27228.018,E2 -27228.018} C_VEL
LIN {X 0,Y 85.628,Z 289.165,A -85,B 0,C 180,E1 -27232.806,E2 -27232.806} C_VEL
LIN {X 0,Y 85.254,Z 286.729,A -85,B 0,C 180,E1 -27236.454,E2 -27236.454} C_VEL
LIN {X 0,Y 85.446,Z 285.851,A -85,B 0,C 180,E1 -27237.654,E2 -27237.654} C_VEL
LIN {X 0,Y 87.671,Z 279.849,A -85,B 0,C 180,E1 -27244.692,E2 -27244.692} C_VEL
LIN {X 0,Y 90.549,Z 272.968,A -85,B 0,C 180,E1 -27250.885,E2 -27250.885} C_VEL
LIN {X 0,Y 94.678,Z 263.756,A -85,B 0,C 180,E1 -27257.132,E2 -27257.132} C_VEL
LIN {X 0,Y 98.661,Z 254.628,A -85,B 0,C 180,E1 -27261.809,E2 -27261.809} C_VEL
LIN {X 0,Y 101.888,Z 246.551,A -85,B 0,C 180,E1 -27265.053,E2 -27265.053} C_VEL
LIN {X 0,Y 101.451,Z 237.277,A -85,B 0,C 180,E1 -27269.333,E2 -27269.333} C_VEL
LIN {X 0,Y 100.09,Z 230.329,A -85,B 0,C 180,E1 -27272.575,E2 -27272.575} C_VEL
LIN {X 0,Y 97.749,Z 222.336,A -85,B 0,C 180,E1 -27276.398,E2 -27276.398} C_VEL
LIN {X 0,Y 93.258,Z 213.146,A -85,B 0,C 180,E1 -27281.578,E2 -27281.578} C_VEL
LIN {X 0,Y 91.792,Z 210.209,A -85,B 0,C 180,E1 -27283.278,E2 -27283.278} C_VEL
LIN {X 0,Y 90.408,Z 208.331,A -85,B 0,C 180,E1 -27284.636,E2 -27284.636} C_VEL
LIN {X 0,Y 89.136,Z 206.061,A -85,B 0,C 180,E1 -27286.073,E2 -27286.073} C_VEL
LIN {X 0,Y 87.264,Z 203.67,A -85,B 0,C 180,E1 -27287.983,E2 -27287.983} C_VEL
LIN {X 0,Y 86.653,Z 201.688,A -85,B 0,C 180,E1 -27289.083,E2 -27289.083} C_VEL
LIN {X 0,Y 86.58,Z 201.687,A -85,B 0,C 180,E1 -27296.764,E2 -27296.764} C_VEL
LIN {X 0,Y 86.501,Z 201.69,A -85,B 0,C 180,E1 -27305.666,E2 -27305.666} C_VEL
LIN {X 0,Y 86.473,Z 201.713,A -85,B 0,C 180,E1 -27312.994,E2 -27312.994} C_VEL
LIN {X 0,Y 86.457,Z 201.692,A -85,B 0,C 180,E1 -27319.438,E2 -27319.438} C_VEL
LIN {X 0,Y 86.533,Z 201.704,A -85,B 0,C 180,E1 -27325.356,E2 -27325.356} C_VEL
LIN {X 0,Y 86.582,Z 201.678,A -85,B 0,C 180,E1 -27333.237,E2 -27333.237} C_VEL
LIN {X 0,Y 86.668,Z 201.677,A -85,B 0,C 180,E1 -27341.076,E2 -27341.076} C_VEL
LIN {X 0,Y 86.93,Z 201.631,A -85,B 0,C 180,E1 -27345.966,E2 -27345.966} C_VEL
LIN {X 0,Y 87.085,Z 201.638,A -85,B 0,C 180,E1 -27350.714,E2 -27350.714} C_VEL
LIN {X 0,Y 87.704,Z 201.546,A -85,B 0,C 180,E1 -27360.002,E2 -27360.002} C_VEL
LIN {X 0,Y 87.084,Z 201.618,A -85,B 0,C 180,E1 -27369.291,E2 -27369.291} C_VEL
LIN {X 0,Y 86.932,Z 201.657,A -85,B 0,C 180,E1 -27374.039,E2 -27374.039} C_VEL
LIN {X 0,Y 86.756,Z 201.73,A -85,B 0,C 180,E1 -27383.896,E2 -27383.896} C_VEL
LIN {X 0,Y 87.816,Z 204.743,A -85,B 0,C 180,E1 -27385.281,E2 -27385.281} C_VEL
LIN {X 0,Y 89.526,Z 207.578,A -85,B 0,C 180,E1 -27387.065,E2 -27387.065} C_VEL
LIN {X 0,Y 91.172,Z 211.396,A -85,B 0,C 180,E1 -27388.962,E2 -27388.962} C_VEL
LIN {X 0,Y 95.557,Z 222.4,A -85,B 0,C 180,E1 -27394.114,E2 -27394.114} C_VEL
LIN {X 0,Y 98.448,Z 231.917,A -85,B 0,C 180,E1 -27398.256,E2 -27398.256} C_VEL
LIN {X 0,Y 99.357,Z 236.382,A -85,B 0,C 180,E1 -27400.089,E2 -27400.089} C_VEL
LIN {X 0,Y 98.805,Z 247.461,A -85,B 0,C 180,E1 -27404.033,E2 -27404.033} C_VEL
LIN {X 0,Y 97.746,Z 257.832,A -85,B 0,C 180,E1 -27408.356,E2 -27408.356} C_VEL
LIN {X 0,Y 96.539,Z 267.559,A -85,B 0,C 180,E1 -27413.21,E2 -27413.21} C_VEL
LIN {X 0,Y 95.481,Z 271.263,A -85,B 0,C 180,E1 -27415.219,E2 -27415.219} C_VEL
LIN {X 0,Y 91.234,Z 280.73,A -85,B 0,C 180,E1 -27421.22,E2 -27421.22} C_VEL
LIN {X 0,Y 87.915,Z 288.3,A -85,B 0,C 180,E1 -27427.684,E2 -27427.684} C_VEL
LIN {X 0,Y 85.528,Z 295.253,A -85,B 0,C 180,E1 -27435.729,E2 -27435.729} C_VEL
LIN {X 0,Y 84.705,Z 299.862,A -85,B 0,C 180,E1 -27442.854,E2 -27442.854} C_VEL
LIN {X 0,Y 84.699,Z 303.307,A -85,B 0,C 180,E1 -27450.001,E2 -27450.001} C_VEL
LIN {X 0,Y 84.492,Z 304.954,A -85,B 0,C 180,E1 -27454.772,E2 -27454.772} C_VEL
LIN {X 0,Y 85.19,Z 307.029,A -85,B 0,C 180,E1 -27464.33,E2 -27464.33} C_VEL
LIN {X 0,Y 88.034,Z 307.647,A -85,B 0,C 180,E1 -27473.527,E2 -27473.527} C_VEL
LIN {X 0,Y 93.222,Z 306.929,A -85,B 0,C 180,E1 -27481.853,E2 -27481.853} C_VEL
LIN {X 0,Y 100.252,Z 304.832,A -85,B 0,C 180,E1 -27489.12,E2 -27489.12} C_VEL
LIN {X 0,Y 108.712,Z 301.288,A -85,B 0,C 180,E1 -27495.328,E2 -27495.328} C_VEL
LIN {X 0,Y 115.893,Z 297.645,A -85,B 0,C 180,E1 -27499.292,E2 -27499.292} C_VEL
LIN {X 0,Y 123.57,Z 293.07,A -85,B 0,C 180,E1 -27502.774,E2 -27502.774} C_VEL
LIN {X 0,Y 128.136,Z 289.642,A -85,B 0,C 180,E1 -27505.359,E2 -27505.359} C_VEL
LIN {X 0,Y 130.433,Z 287.737,A -85,B 0,C 180,E1 -27506.817,E2 -27506.817} C_VEL
LIN {X 0,Y 131.696,Z 286.16,A -85,B 0,C 180,E1 -27508.634,E2 -27508.634} C_VEL
LIN {X 0,Y 132.511,Z 284.541,A -85,B 0,C 180,E1 -27511.487,E2 -27511.487} C_VEL
LIN {X 0,Y 133.142,Z 283.086,A -85,B 0,C 180,E1 -27515.019,E2 -27515.019} C_VEL
LIN {X 0,Y 133.472,Z 282.217,A -85,B 0,C 180,E1 -27518.37,E2 -27518.37} C_VEL
LIN {X 0,Y 133.789,Z 281.735,A -85,B 0,C 180,E1 -27521.627,E2 -27521.627} C_VEL
LIN {X 0,Y 134.026,Z 281.687,A -85,B 0,C 180,E1 -27524.799,E2 -27524.799} C_VEL
LIN {X 0,Y 133.882,Z 282.134,A -85,B 0,C 180,E1 -27527.877,E2 -27527.877} C_VEL
LIN {X 0,Y 133.154,Z 283.242,A -85,B 0,C 180,E1 -27530.888,E2 -27530.888} C_VEL
LIN {X 0,Y 132.45,Z 284.046,A -85,B 0,C 180,E1 -27532.375,E2 -27532.375} C_VEL
LIN {X 0,Y 124.762,Z 288.861,A -85,B 0,C 180,E1 -27535.414,E2 -27535.414} C_VEL
LIN {X 0,Y 115.173,Z 293.749,A -85,B 0,C 180,E1 -27539.998,E2 -27539.998} C_VEL
LIN {X 0,Y 105.952,Z 297.326,A -85,B 0,C 180,E1 -27545.737,E2 -27545.737} C_VEL
LIN {X 0,Y 98.1,Z 299.244,A -85,B 0,C 180,E1 -27552.409,E2 -27552.409} C_VEL
LIN {X 0,Y 93.659,Z 299.751,A -85,B 0,C 180,E1 -27557.464,E2 -27557.464} C_VEL
LIN {X 0,Y 89.996,Z 299.543,A -85,B 0,C 180,E1 -27562.981,E2 -27562.981} C_VEL
LIN {X 0,Y 87.148,Z 298.682,A -85,B 0,C 180,E1 -27568.936,E2 -27568.936} C_VEL
LIN {X 0,Y 84.549,Z 296.146,A -85,B 0,C 180,E1 -27578.249,E2 -27578.249} C_VEL
LIN {X 0,Y 84.031,Z 291.927,A -85,B 0,C 180,E1 -27588.002,E2 -27588.002} C_VEL
LIN {X 0,Y 85.035,Z 287.238,A -85,B 0,C 180,E1 -27595.734,E2 -27595.734} C_VEL
LIN {X 0,Y 85.446,Z 285.851,A -85,B 0,C 180,E1 -27597.654,E2 -27597.654} C_VEL
LIN {X 0,Y 85.731,Z 283.135,A -85,B 0,C 180,E1 -27601.16,E2 -27601.16} C_VEL
LIN {X 0,Y 84.884,Z 278.11,A -85,B 0,C 180,E1 -27606.881,E2 -27606.881} C_VEL
LIN {X 0,Y 84.601,Z 272.47,A -85,B 0,C 180,E1 -27612.433,E2 -27612.433} C_VEL
LIN {X 0,Y 85.729,Z 268.706,A -85,B 0,C 180,E1 -27615.452,E2 -27615.452} C_VEL
LIN {X 0,Y 89.896,Z 259.887,A -85,B 0,C 180,E1 -27621.004,E2 -27621.004} C_VEL
LIN {X 0,Y 94.272,Z 249.95,A -85,B 0,C 180,E1 -27625.724,E2 -27625.724} C_VEL
LIN {X 0,Y 95.319,Z 247.211,A -85,B 0,C 180,E1 -27626.829,E2 -27626.829} C_VEL
LIN {X 0,Y 95.016,Z 238.447,A -85,B 0,C 180,E1 -27631.187,E2 -27631.187} C_VEL
LIN {X 0,Y 93.799,Z 232.532,A -85,B 0,C 180,E1 -27634.296,E2 -27634.296} C_VEL
LIN {X 0,Y 91.724,Z 225.219,A -85,B 0,C 180,E1 -27638.224,E2 -27638.224} C_VEL
LIN {X 0,Y 87.488,Z 216.185,A -85,B 0,C 180,E1 -27643.944,E2 -27643.944} C_VEL
LIN {X 0,Y 85.068,Z 211.693,A -85,B 0,C 180,E1 -27647.107,E2 -27647.107} C_VEL
LIN {X 0,Y 82.872,Z 208.516,A -85,B 0,C 180,E1 -27649.829,E2 -27649.829} C_VEL
LIN {X 0,Y 82.127,Z 207.16,A -85,B 0,C 180,E1 -27650.896,E2 -27650.896} C_VEL
LIN {X 0,Y 80.221,Z 204.844,A -85,B 0,C 180,E1 -27653.256,E2 -27653.256} C_VEL
LIN {X 0,Y 79.544,Z 202.567,A -85,B 0,C 180,E1 -27654.812,E2 -27654.812} C_VEL
LIN {X 0,Y 79.372,Z 202.6,A -85,B 0,C 180,E1 -27662.09,E2 -27662.09} C_VEL
LIN {X 0,Y 79.361,Z 202.582,A -85,B 0,C 180,E1 -27668.308,E2 -27668.308} C_VEL
LIN {X 0,Y 79.383,Z 202.584,A -85,B 0,C 180,E1 -27675.093,E2 -27675.093} C_VEL
LIN {X 0,Y 79.386,Z 202.592,A -85,B 0,C 180,E1 -27682.821,E2 -27682.821} C_VEL
LIN {X 0,Y 79.378,Z 202.583,A -85,B 0,C 180,E1 -27687.914,E2 -27687.914} C_VEL
LIN {X 0,Y 79.523,Z 202.559,A -85,B 0,C 180,E1 -27693.779,E2 -27693.779} C_VEL
LIN {X 0,Y 79.526,Z 202.576,A -85,B 0,C 180,E1 -27699.302,E2 -27699.302} C_VEL
LIN {X 0,Y 79.824,Z 202.514,A -85,B 0,C 180,E1 -27705.575,E2 -27705.575} C_VEL
LIN {X 0,Y 79.967,Z 202.522,A -85,B 0,C 180,E1 -27709.879,E2 -27709.879} C_VEL
LIN {X 0,Y 80.633,Z 202.425,A -85,B 0,C 180,E1 -27720.003,E2 -27720.003} C_VEL
LIN {X 0,Y 79.967,Z 202.506,A -85,B 0,C 180,E1 -27730.126,E2 -27730.126} C_VEL
LIN {X 0,Y 79.752,Z 202.547,A -85,B 0,C 180,E1 -27735.332,E2 -27735.332} C_VEL
LIN {X 0,Y 79.684,Z 202.728,A -85,B 0,C 180,E1 -27738.316,E2 -27738.316} C_VEL
LIN {X 0,Y 80.634,Z 205.425,A -85,B 0,C 180,E1 -27739.908,E2 -27739.908} C_VEL
LIN {X 0,Y 82.868,Z 208.039,A -85,B 0,C 180,E1 -27742.438,E2 -27742.438} C_VEL
LIN {X 0,Y 85.148,Z 212.956,A -85,B 0,C 180,E1 -27745.479,E2 -27745.479} C_VEL
LIN {X 0,Y 88.475,Z 221.49,A -85,B 0,C 180,E1 -27750.18,E2 -27750.18} C_VEL
LIN {X 0,Y 91.315,Z 230.293,A -85,B 0,C 180,E1 -27754.586,E2 -27754.586} C_VEL
LIN {X 0,Y 93.105,Z 237.853,A -85,B 0,C 180,E1 -27758.162,E2 -27758.162} C_VEL
LIN {X 0,Y 92.318,Z 249.007,A -85,B 0,C 180,E1 -27762.579,E2 -27762.579} C_VEL
LIN {X 0,Y 90.935,Z 259.605,A -85,B 0,C 180,E1 -27767.45,E2 -27767.45} C_VEL
LIN {X 0,Y 89.511,Z 268.906,A -85,B 0,C 180,E1 -27772.593,E2 -27772.593} C_VEL
LIN {X 0,Y 87.258,Z 274.081,A -85,B 0,C 180,E1 -27775.682,E2 -27775.682} C_VEL
LIN {X 0,Y 83.137,Z 282.874,A -85,B 0,C 180,E1 -27782.294,E2 -27782.294} C_VEL
LIN {X 0,Y 79.999,Z 289.933,A -85,B 0,C 180,E1 -27789.428,E2 -27789.428} C_VEL
LIN {X 0,Y 78.213,Z 295.605,A -85,B 0,C 180,E1 -27797.019,E2 -27797.019} C_VEL
LIN {X 0,Y 77.63,Z 300.028,A -85,B 0,C 180,E1 -27804.807,E2 -27804.807} C_VEL
LIN {X 0,Y 77.653,Z 302.305,A -85,B 0,C 180,E1 -27810.001,E2 -27810.001} C_VEL
LIN {X 0,Y 77.476,Z 304.037,A -85,B 0,C 180,E1 -27815.205,E2 -27815.205} C_VEL
LIN {X 0,Y 78.343,Z 306.305,A -85,B 0,C 180,E1 -27825.613,E2 -27825.613} C_VEL
LIN {X 0,Y 81.552,Z 307.162,A -85,B 0,C 180,E1 -27835.525,E2 -27835.525} C_VEL
LIN {X 0,Y 87.245,Z 306.637,A -85,B 0,C 180,E1 -27844.326,E2 -27844.326} C_VEL
LIN {X 0,Y 94.833,Z 304.773,A -85,B 0,C 180,E1 -27851.836,E2 -27851.836} C_VEL
LIN {X 0,Y 103.841,Z 301.521,A -85,B 0,C 180,E1 -27858.116,E2 -27858.116} C_VEL
LIN {X 0,Y 114.055,Z 296.734,A -85,B 0,C 180,E1 -27863.232,E2 -27863.232} C_VEL
LIN {X 0,Y 119.38,Z 293.767,A -85,B 0,C 180,E1 -27865.508,E2 -27865.508} C_VEL
LIN {X 0,Y 124.127,Z 290.542,A -85,B 0,C 180,E1 -27868.136,E2 -27868.136} C_VEL
LIN {X 0,Y 125.674,Z 289.114,A -85,B 0,C 180,E1 -27869.78,E2 -27869.78} C_VEL
LIN {X 0,Y 126.779,Z 287.332,A -85,B 0,C 180,E1 -27873.672,E2 -27873.672} C_VEL
LIN {X 0,Y 127.262,Z 286.293,A -85,B 0,C 180,E1 -27877.257,E2 -27877.257} C_VEL
LIN {X 0,Y 127.676,Z 285.668,A -85,B 0,C 180,E1 -27880.713,E2 -27880.713} C_VEL
LIN {X 0,Y 127.922,Z 285.445,A -85,B 0,C 180,E1 -27884.054,E2 -27884.054} C_VEL
LIN {X 0,Y 127.817,Z 285.728,A -85,B 0,C 180,E1 -27887.293,E2 -27887.293} C_VEL
LIN {X 0,Y 126.937,Z 286.697,A -85,B 0,C 180,E1 -27890.437,E2 -27890.437} C_VEL
LIN {X 0,Y 116.081,Z 292.473,A -85,B 0,C 180,E1 -27894.714,E2 -27894.714} C_VEL
LIN {X 0,Y 105.422,Z 296.762,A -85,B 0,C 180,E1 -27900.138,E2 -27900.138} C_VEL
LIN {X 0,Y 98.705,Z 298.724,A -85,B 0,C 180,E1 -27904.552,E2 -27904.552} C_VEL
LIN {X 0,Y 92.667,Z 299.859,A -85,B 0,C 180,E1 -27909.613,E2 -27909.613} C_VEL
LIN {X 0,Y 87.44,Z 300.231,A -85,B 0,C 180,E1 -27915.309,E2 -27915.309} C_VEL
LIN {X 0,Y 83.182,Z 299.846,A -85,B 0,C 180,E1 -27921.658,E2 -27921.658} C_VEL
LIN {X 0,Y 79.98,Z 298.679,A -85,B 0,C 180,E1 -27928.51,E2 -27928.51} C_VEL
LIN {X 0,Y 77.879,Z 296.741,A -85,B 0,C 180,E1 -27935.688,E2 -27935.688} C_VEL
LIN {X 0,Y 76.914,Z 294.061,A -85,B 0,C 180,E1 -27943.028,E2 -27943.028} C_VEL
LIN {X 0,Y 77.344,Z 289.32,A -85,B 0,C 180,E1 -27952.628,E2 -27952.628} C_VEL
LIN {X 0,Y 78.842,Z 284.461,A -85,B 0,C 180,E1 -27959.969,E2 -27959.969} C_VEL
LIN {X 0,Y 81.267,Z 278.442,A -85,B 0,C 180,E1 -27967.037,E2 -27967.037} C_VEL
LIN {X 0,Y 85.07,Z 270.11,A -85,B 0,C 180,E1 -27974.424,E2 -27974.424} C_VEL
LIN {X 0,Y 85.729,Z 268.706,A -85,B 0,C 180,E1 -27975.452,E2 -27975.452} C_VEL
LIN {X 0,Y 87.183,Z 264.786,A -85,B 0,C 180,E1 -27978.233,E2 -27978.233} C_VEL
LIN {X 0,Y 88.024,Z 260.687,A -85,B 0,C 180,E1 -27980.999,E2 -27980.999} C_VEL
LIN {X 0,Y 88.343,Z 257.884,A -85,B 0,C 180,E1 -27982.819,E2 -27982.819} C_VEL
LIN {X 0,Y 88.658,Z 252.088,A -85,B 0,C 180,E1 -27986.406,E2 -27986.406} C_VEL
LIN {X 0,Y 88.877,Z 246.036,A -85,B 0,C 180,E1 -27989.808,E2 -27989.808} C_VEL
LIN {X 0,Y 88.622,Z 239.718,A -85,B 0,C 180,E1 -27993.252,E2 -27993.252} C_VEL
LIN {X 0,Y 86.695,Z 230.647,A -85,B 0,C 180,E1 -27998.581,E2 -27998.581} C_VEL
LIN {X 0,Y 82.984,Z 221.719,A -85,B 0,C 180,E1 -28004.718,E2 -28004.718} C_VEL
LIN {X 0,Y 80.778,Z 217.303,A -85,B 0,C 180,E1 -28008.181,E2 -28008.181} C_VEL
LIN {X 0,Y 78.182,Z 212.872,A -85,B 0,C 180,E1 -28012.159,E2 -28012.159} C_VEL
LIN {X 0,Y 76.889,Z 211.343,A -85,B 0,C 180,E1 -28013.936,E2 -28013.936} C_VEL
LIN {X 0,Y 75.563,Z 208.438,A -85,B 0,C 180,E1 -28016.476,E2 -28016.476} C_VEL
LIN {X 0,Y 73.169,Z 206.054,A -85,B 0,C 180,E1 -28020.184,E2 -28020.184} C_VEL
LIN {X 0,Y 72.32,Z 203.475,A -85,B 0,C 180,E1 -28022.511,E2 -28022.511} C_VEL
LIN {X 0,Y 72.29,Z 203.466,A -85,B 0,C 180,E1 -28028.949,E2 -28028.949} C_VEL
LIN {X 0,Y 72.243,Z 203.46,A -85,B 0,C 180,E1 -28037.084,E2 -28037.084} C_VEL
LIN {X 0,Y 72.293,Z 203.479,A -85,B 0,C 180,E1 -28044.321,E2 -28044.321} C_VEL
LIN {X 0,Y 72.372,Z 203.439,A -85,B 0,C 180,E1 -28050.955,E2 -28050.955} C_VEL
LIN {X 0,Y 72.4,Z 203.465,A -85,B 0,C 180,E1 -28057.155,E2 -28057.155} C_VEL
LIN {X 0,Y 72.743,Z 203.393,A -85,B 0,C 180,E1 -28065.044,E2 -28065.044} C_VEL
LIN {X 0,Y 72.858,Z 203.402,A -85,B 0,C 180,E1 -28068.879,E2 -28068.879} C_VEL
LIN {X 0,Y 73.561,Z 203.304,A -85,B 0,C 180,E1 -28080.003,E2 -28080.003} C_VEL
LIN {X 0,Y 72.893,Z 203.575,A -85,B 0,C 180,E1 -28091.121,E2 -28091.121} C_VEL
LIN {X 0,Y 73.728,Z 206.147,A -85,B 0,C 180,E1 -28093.045,E2 -28093.045} C_VEL
LIN {X 0,Y 76.054,Z 209.025,A -85,B 0,C 180,E1 -28096.615,E2 -28096.615} C_VEL
LIN {X 0,Y 77.799,Z 212.266,A -85,B 0,C 180,E1 -28099.461,E2 -28099.461} C_VEL
LIN {X 0,Y 78.869,Z 213.699,A -85,B 0,C 180,E1 -28100.885,E2 -28100.885} C_VEL
LIN {X 0,Y 81.666,Z 220.631,A -85,B 0,C 180,E1 -28105.489,E2 -28105.489} C_VEL
LIN {X 0,Y 84.756,Z 230.411,A -85,B 0,C 180,E1 -28111.218,E2 -28111.218} C_VEL
LIN {X 0,Y 86.904,Z 239.989,A -85,B 0,C 180,E1 -28116.337,E2 -28116.337} C_VEL
LIN {X 0,Y 85.904,Z 250.464,A -85,B 0,C 180,E1 -28120.885,E2 -28120.885} C_VEL
LIN {X 0,Y 84.357,Z 260.163,A -85,B 0,C 180,E1 -28125.755,E2 -28125.755} C_VEL
LIN {X 0,Y 82.863,Z 268.606,A -85,B 0,C 180,E1 -28130.843,E2 -28130.843} C_VEL
LIN {X 0,Y 81.507,Z 271.82,A -85,B 0,C 180,E1 -28132.874,E2 -28132.874} C_VEL
LIN {X 0,Y 77.602,Z 279.595,A -85,B 0,C 180,E1 -28138.619,E2 -28138.619} C_VEL
LIN {X 0,Y 73.888,Z 287.216,A -85,B 0,C 180,E1 -28146.157,E2 -28146.157} C_VEL
LIN {X 0,Y 71.347,Z 294.182,A -85,B 0,C 180,E1 -28155.745,E2 -28155.745} C_VEL
LIN {X 0,Y 70.604,Z 298.917,A -85,B 0,C 180,E1 -28164.54,E2 -28164.54} C_VEL
LIN {X 0,Y 70.611,Z 301.224,A -85,B 0,C 180,E1 -28170.001,E2 -28170.001} C_VEL
LIN {X 0,Y 70.446,Z 303.083,A -85,B 0,C 180,E1 -28175.727,E2 -28175.727} C_VEL
LIN {X 0,Y 71.546,Z 305.542,A -85,B 0,C 180,E1 -28187.14,E2 -28187.14} C_VEL
LIN {X 0,Y 75.19,Z 306.599,A -85,B 0,C 180,E1 -28197.863,E2 -28197.863} C_VEL
LIN {X 0,Y 81.457,Z 306.343,A -85,B 0,C 180,E1 -28207.155,E2 -28207.155} C_VEL
LIN {X 0,Y 89.656,Z 304.694,A -85,B 0,C 180,E1 -28214.871,E2 -28214.871} C_VEL
LIN {X 0,Y 99.23,Z 301.695,A -85,B 0,C 180,E1 -28221.178,E2 -28221.178} C_VEL
LIN {X 0,Y 109.963,Z 297.252,A -85,B 0,C 180,E1 -28226.188,E2 -28226.188} C_VEL
LIN {X 0,Y 112.802,Z 295.858,A -85,B 0,C 180,E1 -28227.258,E2 -28227.258} C_VEL
LIN {X 0,Y 115.464,Z 294.432,A -85,B 0,C 180,E1 -28228.447,E2 -28228.447} C_VEL
LIN {X 0,Y 117.964,Z 292.944,A -85,B 0,C 180,E1 -28229.756,E2 -28229.756} C_VEL
LIN {X 0,Y 119.87,Z 291.424,A -85,B 0,C 180,E1 -28232.026,E2 -28232.026} C_VEL
LIN {X 0,Y 120.761,Z 290.072,A -85,B 0,C 180,E1 -28235.958,E2 -28235.958} C_VEL
LIN {X 0,Y 121.316,Z 289.292,A -85,B 0,C 180,E1 -28239.658,E2 -28239.658} C_VEL
LIN {X 0,Y 121.599,Z 288.924,A -85,B 0,C 180,E1 -28243.201,E2 -28243.201} C_VEL
LIN {X 0,Y 121.574,Z 289.043,A -85,B 0,C 180,E1 -28246.629,E2 -28246.629} C_VEL
LIN {X 0,Y 121.116,Z 289.409,A -85,B 0,C 180,E1 -28248.28,E2 -28248.28} C_VEL
LIN {X 0,Y 113.808,Z 292.924,A -85,B 0,C 180,E1 -28251.138,E2 -28251.138} C_VEL
LIN {X 0,Y 102.868,Z 297.116,A -85,B 0,C 180,E1 -28256.08,E2 -28256.08} C_VEL
LIN {X 0,Y 96.11,Z 298.963,A -85,B 0,C 180,E1 -28259.998,E2 -28259.998} C_VEL
LIN {X 0,Y 89.853,Z 300.157,A -85,B 0,C 180,E1 -28264.484,E2 -28264.484} C_VEL
LIN {X 0,Y 84.241,Z 300.706,A -85,B 0,C 180,E1 -28269.602,E2 -28269.602} C_VEL
LIN {X 0,Y 79.401,Z 300.562,A -85,B 0,C 180,E1 -28275.396,E2 -28275.396} C_VEL
LIN {X 0,Y 75.455,Z 299.795,A -85,B 0,C 180,E1 -28281.871,E2 -28281.871} C_VEL
LIN {X 0,Y 71.344,Z 297.287,A -85,B 0,C 180,E1 -28292.799,E2 -28292.799} C_VEL
LIN {X 0,Y 69.935,Z 294.524,A -85,B 0,C 180,E1 -28301.091,E2 -28301.091} C_VEL
LIN {X 0,Y 70.08,Z 290.039,A -85,B 0,C 180,E1 -28311.189,E2 -28311.189} C_VEL
LIN {X 0,Y 71.824,Z 284.348,A -85,B 0,C 180,E1 -28320.707,E2 -28320.707} C_VEL
LIN {X 0,Y 74.96,Z 277.072,A -85,B 0,C 180,E1 -28329.639,E2 -28329.639} C_VEL
LIN {X 0,Y 79.221,Z 268.396,A -85,B 0,C 180,E1 -28337.371,E2 -28337.371} C_VEL
LIN {X 0,Y 83.979,Z 258.752,A -85,B 0,C 180,E1 -28343.617,E2 -28343.617} C_VEL
LIN {X 0,Y 88.506,Z 248.945,A -85,B 0,C 180,E1 -28348.293,E2 -28348.293} C_VEL
LIN {X 0,Y 88.877,Z 246.036,A -85,B 0,C 180,E1 -28349.808,E2 -28349.808} C_VEL
LIN {X 0,Y 88.605,Z 243.13,A -85,B 0,C 180,E1 -28351.491,E2 -28351.491} C_VEL
LIN {X 0,Y 87.673,Z 240.504,A -85,B 0,C 180,E1 -28353.292,E2 -28353.292} C_VEL
LIN {X 0,Y 85.505,Z 237.003,A -85,B 0,C 180,E1 -28356.16,E2 -28356.16} C_VEL
LIN {X 0,Y 79.473,Z 229.357,A -85,B 0,C 180,E1 -28363.562,E2 -28363.562} C_VEL
LIN {X 0,Y 78.176,Z 226.834,A -85,B 0,C 180,E1 -28365.747,E2 -28365.747} C_VEL
LIN {X 0,Y 75.884,Z 221.924,A -85,B 0,C 180,E1 -28370.049,E2 -28370.049} C_VEL
LIN {X 0,Y 73.51,Z 217.676,A -85,B 0,C 180,E1 -28374.383,E2 -28374.383} C_VEL
LIN {X 0,Y 71.729,Z 214.179,A -85,B 0,C 180,E1 -28378.144,E2 -28378.144} C_VEL
LIN {X 0,Y 69.526,Z 211.495,A -85,B 0,C 180,E1 -28382.377,E2 -28382.377} C_VEL
LIN {X 0,Y 68.554,Z 209.486,A -85,B 0,C 180,E1 -28384.906,E2 -28384.906} C_VEL
LIN {X 0,Y 65.801,Z 206.501,A -85,B 0,C 180,E1 -28391.618,E2 -28391.618} C_VEL
LIN {X 0,Y 65.156,Z 204.354,A -85,B 0,C 180,E1 -28394.855,E2 -28394.855} C_VEL
LIN {X 0,Y 65.199,Z 204.338,A -85,B 0,C 180,E1 -28399.707,E2 -28399.707} C_VEL
LIN {X 0,Y 65.252,Z 204.328,A -85,B 0,C 180,E1 -28409.5,E2 -28409.5} C_VEL
LIN {X 0,Y 65.24,Z 204.34,A -85,B 0,C 180,E1 -28414.479,E2 -28414.479} C_VEL
LIN {X 0,Y 65.641,Z 204.277,A -85,B 0,C 180,E1 -28424.492,E2 -28424.492} C_VEL
LIN {X 0,Y 65.763,Z 204.274,A -85,B 0,C 180,E1 -28427.662,E2 -28427.662} C_VEL
LIN {X 0,Y 66.486,Z 204.184,A -85,B 0,C 180,E1 -28440.003,E2 -28440.003} C_VEL
LIN {X 0,Y 66.402,Z 204.519,A -85,B 0,C 180,E1 -28440.951,E2 -28440.951} C_VEL
LIN {X 0,Y 66.992,Z 206.88,A -85,B 0,C 180,E1 -28443.386,E2 -28443.386} C_VEL
LIN {X 0,Y 68.817,Z 209.141,A -85,B 0,C 180,E1 -28447.706,E2 -28447.706} C_VEL
LIN {X 0,Y 69.529,Z 209.806,A -85,B 0,C 180,E1 -28449.09,E2 -28449.09} C_VEL
LIN {X 0,Y 70.963,Z 212.904,A -85,B 0,C 180,E1 -28452.396,E2 -28452.396} C_VEL
LIN {X 0,Y 72.089,Z 214.218,A -85,B 0,C 180,E1 -28454.308,E2 -28454.308} C_VEL
LIN {X 0,Y 75.014,Z 219.917,A -85,B 0,C 180,E1 -28459.857,E2 -28459.857} C_VEL
LIN {X 0,Y 77.486,Z 227.677,A -85,B 0,C 180,E1 -28465.345,E2 -28465.345} C_VEL
LIN {X 0,Y 79.255,Z 234.237,A -85,B 0,C 180,E1 -28469.558,E2 -28469.558} C_VEL
LIN {X 0,Y 80.745,Z 242.076,A -85,B 0,C 180,E1 -28474.284,E2 -28474.284} C_VEL
LIN {X 0,Y 79.542,Z 251.588,A -85,B 0,C 180,E1 -28478.875,E2 -28478.875} C_VEL
LIN {X 0,Y 77.488,Z 262.149,A -85,B 0,C 180,E1 -28484.779,E2 -28484.779} C_VEL
LIN {X 0,Y 75.91,Z 269.388,A -85,B 0,C 180,E1 -28489.604,E2 -28489.604} C_VEL
LIN {X 0,Y 70.889,Z 278.931,A -85,B 0,C 180,E1 -28496.958,E2 -28496.958} C_VEL
LIN {X 0,Y 66.926,Z 286.568,A -85,B 0,C 180,E1 -28505.164,E2 -28505.164} C_VEL
LIN {X 0,Y 64.504,Z 292.696,A -85,B 0,C 180,E1 -28514.195,E2 -28514.195} C_VEL
LIN {X 0,Y 63.561,Z 297.845,A -85,B 0,C 180,E1 -28524.378,E2 -28524.378} C_VEL
LIN {X 0,Y 63.576,Z 300.074,A -85,B 0,C 180,E1 -28530.001,E2 -28530.001} C_VEL
LIN {X 0,Y 63.443,Z 302.051,A -85,B 0,C 180,E1 -28536.361,E2 -28536.361} C_VEL
LIN {X 0,Y 64.785,Z 304.754,A -85,B 0,C 180,E1 -28548.994,E2 -28548.994} C_VEL
LIN {X 0,Y 68.979,Z 306.01,A -85,B 0,C 180,E1 -28560.627,E2 -28560.627} C_VEL
LIN {X 0,Y 75.902,Z 305.962,A -85,B 0,C 180,E1 -28570.404,E2 -28570.404} C_VEL
LIN {X 0,Y 84.753,Z 304.599,A -85,B 0,C 180,E1 -28578.273,E2 -28578.273} C_VEL
LIN {X 0,Y 94.938,Z 301.868,A -85,B 0,C 180,E1 -28584.52,E2 -28584.52} C_VEL
LIN {X 0,Y 106.189,Z 297.687,A -85,B 0,C 180,E1 -28589.362,E2 -28589.362} C_VEL
LIN {X 0,Y 109.116,Z 296.433,A -85,B 0,C 180,E1 -28590.404,E2 -28590.404} C_VEL
LIN {X 0,Y 111.844,Z 295.084,A -85,B 0,C 180,E1 -28591.611,E2 -28591.611} C_VEL
LIN {X 0,Y 113.814,Z 293.677,A -85,B 0,C 180,E1 -28594.388,E2 -28594.388} C_VEL
LIN {X 0,Y 114.73,Z 292.625,A -85,B 0,C 180,E1 -28598.434,E2 -28598.434} C_VEL
LIN {X 0,Y 115.092,Z 292.136,A -85,B 0,C 180,E1 -28602.221,E2 -28602.221} C_VEL
LIN {X 0,Y 115.158,Z 292.072,A -85,B 0,C 180,E1 -28605.869,E2 -28605.869} C_VEL
LIN {X 0,Y 112.274,Z 293.328,A -85,B 0,C 180,E1 -28607.343,E2 -28607.343} C_VEL
LIN {X 0,Y 100.639,Z 297.531,A -85,B 0,C 180,E1 -28611.969,E2 -28611.969} C_VEL
LIN {X 0,Y 91.513,Z 299.81,A -85,B 0,C 180,E1 -28616.742,E2 -28616.742} C_VEL
LIN {X 0,Y 84.369,Z 300.884,A -85,B 0,C 180,E1 -28621.574,E2 -28621.574} C_VEL
LIN {X 0,Y 77.935,Z 301.209,A -85,B 0,C 180,E1 -28627.263,E2 -28627.263} C_VEL
LIN {X 0,Y 70.135,Z 300.331,A -85,B 0,C 180,E1 -28637.492,E2 -28637.492} C_VEL
LIN {X 0,Y 66.497,Z 298.867,A -85,B 0,C 180,E1 -28645.005,E2 -28645.005} C_VEL
LIN {X 0,Y 64.008,Z 296.705,A -85,B 0,C 180,E1 -28653.294,E2 -28653.294} C_VEL
LIN {X 0,Y 62.663,Z 292.651,A -85,B 0,C 180,E1 -28664.978,E2 -28664.978} C_VEL
LIN {X 0,Y 63.703,Z 287.199,A -85,B 0,C 180,E1 -28676.52,E2 -28676.52} C_VEL
LIN {X 0,Y 66.141,Z 281.082,A -85,B 0,C 180,E1 -28686.038,E2 -28686.038} C_VEL
LIN {X 0,Y 69.333,Z 274.522,A -85,B 0,C 180,E1 -28693.749,E2 -28693.749} C_VEL
LIN {X 0,Y 74.338,Z 265.074,A -85,B 0,C 180,E1 -28701.846,E2 -28701.846} C_VEL
LIN {X 0,Y 79.057,Z 256.012,A -85,B 0,C 180,E1 -28707.452,E2 -28707.452} C_VEL
LIN {X 0,Y 82.28,Z 249.353,A -85,B 0,C 180,E1 -28710.611,E2 -28710.611} C_VEL
LIN {X 0,Y 82.55,Z 244.167,A -85,B 0,C 180,E1 -28713.66,E2 -28713.66} C_VEL
LIN {X 0,Y 81.952,Z 239.347,A -85,B 0,C 180,E1 -28716.712,E2 -28716.712} C_VEL
LIN {X 0,Y 80.573,Z 232.997,A -85,B 0,C 180,E1 -28720.951,E2 -28720.951} C_VEL
LIN {X 0,Y 78.176,Z 226.834,A -85,B 0,C 180,E1 -28725.747,E2 -28725.747} C_VEL
LIN {X 0,Y 76.178,Z 223.484,A -85,B 0,C 180,E1 -28729.051,E2 -28729.051} C_VEL
LIN {X 0,Y 72.655,Z 220.298,A -85,B 0,C 180,E1 -28733.957,E2 -28733.957} C_VEL
LIN {X 0,Y 64.942,Z 215.275,A -85,B 0,C 180,E1 -28747.217,E2 -28747.217} C_VEL
LIN {X 0,Y 62.946,Z 212.666,A -85,B 0,C 180,E1 -28753.471,E2 -28753.471} C_VEL
LIN {X 0,Y 62.175,Z 210.775,A -85,B 0,C 180,E1 -28757.3,E2 -28757.3} C_VEL
LIN {X 0,Y 59.833,Z 208.991,A -85,B 0,C 180,E1 -28771.98,E2 -28771.98} C_VEL
LIN {X 0,Y 60.355,Z 209.005,A -85,B 0,C 180,E1 -28785.2,E2 -28785.2} C_VEL
LIN {X 0,Y 63.522,Z 210.897,A -85,B 0,C 180,E1 -28798.706,E2 -28798.706} C_VEL
LIN {X 0,Y 64.586,Z 213.953,A -85,B 0,C 180,E1 -28803.122,E2 -28803.122} C_VEL
LIN {X 0,Y 66.26,Z 216.265,A -85,B 0,C 180,E1 -28807.622,E2 -28807.622} C_VEL
LIN {X 0,Y 68.522,Z 220.709,A -85,B 0,C 180,E1 -28813.346,E2 -28813.346} C_VEL
LIN {X 0,Y 70.743,Z 225.395,A -85,B 0,C 180,E1 -28818.357,E2 -28818.357} C_VEL
LIN {X 0,Y 73.101,Z 234.911,A -85,B 0,C 180,E1 -28825.638,E2 -28825.638} C_VEL
LIN {X 0,Y 74.501,Z 243.13,A -85,B 0,C 180,E1 -28831.261,E2 -28831.261} C_VEL
LIN {X 0,Y 74.692,Z 244.442,A -85,B 0,C 180,E1 -28832.132,E2 -28832.132} C_VEL
LIN {X 0,Y 72.844,Z 254.729,A -85,B 0,C 180,E1 -28837.684,E2 -28837.684} C_VEL
LIN {X 0,Y 70.497,Z 264.909,A -85,B 0,C 180,E1 -28844.258,E2 -28844.258} C_VEL
LIN {X 0,Y 69.549,Z 268.599,A -85,B 0,C 180,E1 -28846.993,E2 -28846.993} C_VEL
LIN {X 0,Y 65.891,Z 275.268,A -85,B 0,C 180,E1 -28852.173,E2 -28852.173} C_VEL
LIN {X 0,Y 61.927,Z 282.275,A -85,B 0,C 180,E1 -28859.291,E2 -28859.291} C_VEL
LIN {X 0,Y 58.471,Z 289.17,A -85,B 0,C 180,E1 -28868.865,E2 -28868.865} C_VEL
LIN {X 0,Y 56.77,Z 294.671,A -85,B 0,C 180,E1 -28879.3,E2 -28879.3} C_VEL
LIN {X 0,Y 56.543,Z 298.902,A -85,B 0,C 180,E1 -28890.001,E2 -28890.001} C_VEL
LIN {X 0,Y 56.457,Z 300.965,A -85,B 0,C 180,E1 -28897.152,E2 -28897.152} C_VEL
LIN {X 0,Y 58.144,Z 303.871,A -85,B 0,C 180,E1 -28911.262,E2 -28911.262} C_VEL
LIN {X 0,Y 62.962,Z 305.39,A -85,B 0,C 180,E1 -28923.927,E2 -28923.927} C_VEL
LIN {X 0,Y 70.629,Z 305.581,A -85,B 0,C 180,E1 -28934.152,E2 -28934.152} C_VEL
LIN {X 0,Y 81.104,Z 304.277,A -85,B 0,C 180,E1 -28942.655,E2 -28942.655} C_VEL
LIN {X 0,Y 90.996,Z 301.984,A -85,B 0,C 180,E1 -28948.167,E2 -28948.167} C_VEL
LIN {X 0,Y 102.764,Z 298.151,A -85,B 0,C 180,E1 -28952.758,E2 -28952.758} C_VEL
LIN {X 0,Y 105.76,Z 296.934,A -85,B 0,C 180,E1 -28953.782,E2 -28953.782} C_VEL
LIN {X 0,Y 107.573,Z 295.903,A -85,B 0,C 180,E1 -28956.159,E2 -28956.159} C_VEL
LIN {X 0,Y 108.382,Z 295.052,A -85,B 0,C 180,E1 -28961.079,E2 -28961.079} C_VEL
LIN {X 0,Y 108.532,Z 294.868,A -85,B 0,C 180,E1 -28963.056,E2 -28963.056} C_VEL
LIN {X 0,Y 107.057,Z 295.354,A -85,B 0,C 180,E1 -28964.774,E2 -28964.774} C_VEL
LIN {X 0,Y 98.957,Z 297.988,A -85,B 0,C 180,E1 -28967.696,E2 -28967.696} C_VEL
LIN {X 0,Y 91.116,Z 299.876,A -85,B 0,C 180,E1 -28971.124,E2 -28971.124} C_VEL
LIN {X 0,Y 83.731,Z 301.104,A -85,B 0,C 180,E1 -28975.183,E2 -28975.183} C_VEL
LIN {X 0,Y 76.849,Z 301.669,A -85,B 0,C 180,E1 -28979.997,E2 -28979.997} C_VEL
LIN {X 0,Y 70.632,Z 301.572,A -85,B 0,C 180,E1 -28985.708,E2 -28985.708} C_VEL
LIN {X 0,Y 64.911,Z 300.767,A -85,B 0,C 180,E1 -28992.975,E2 -28992.975} C_VEL
LIN {X 0,Y 60.406,Z 299.18,A -85,B 0,C 180,E1 -29001.441,E2 -29001.441} C_VEL
LIN {X 0,Y 56.525,Z 295.757,A -85,B 0,C 180,E1 -29014.596,E2 -29014.596} C_VEL
LIN {X 0,Y 55.575,Z 292.159,A -85,B 0,C 180,E1 -29025.272,E2 -29025.272} C_VEL
LIN {X 0,Y 56.747,Z 286.587,A -85,B 0,C 180,E1 -29037.864,E2 -29037.864} C_VEL
LIN {X 0,Y 59.165,Z 281.024,A -85,B 0,C 180,E1 -29047.289,E2 -29047.289} C_VEL
LIN {X 0,Y 63.362,Z 273.045,A -85,B 0,C 180,E1 -29057.182,E2 -29057.182} C_VEL
LIN {X 0,Y 68.404,Z 264.15,A -85,B 0,C 180,E1 -29064.969,E2 -29064.969} C_VEL
LIN {X 0,Y 73.469,Z 254.945,A -85,B 0,C 180,E1 -29070.684,E2 -29070.684} C_VEL
LIN {X 0,Y 76.105,Z 249.64,A -85,B 0,C 180,E1 -29073.308,E2 -29073.308} C_VEL
LIN {X 0,Y 76.246,Z 245.073,A -85,B 0,C 180,E1 -29076.346,E2 -29076.346} C_VEL
LIN {X 0,Y 75.144,Z 237.482,A -85,B 0,C 180,E1 -29081.919,E2 -29081.919} C_VEL
LIN {X 0,Y 72.504,Z 229.845,A -85,B 0,C 180,E1 -29088.604,E2 -29088.604} C_VEL
LIN {X 0,Y 69.748,Z 223.838,A -85,B 0,C 180,E1 -29094.932,E2 -29094.932} C_VEL
LIN {X 0,Y 67.751,Z 219.803,A -85,B 0,C 180,E1 -29099.927,E2 -29099.927} C_VEL
LIN {X 0,Y 64.942,Z 215.275,A -85,B 0,C 180,E1 -29107.217,E2 -29107.217} C_VEL
LIN {X 0,Y 62.98,Z 214.157,A -85,B 0,C 180,E1 -29112.121,E2 -29112.121} C_VEL
LIN {X 0,Y 61.032,Z 214.07,A -85,B 0,C 180,E1 -29117.327,E2 -29117.327} C_VEL
LIN {X 0,Y 57.654,Z 215.599,A -85,B 0,C 180,E1 -29132.576,E2 -29132.576} C_VEL
LIN {X 0,Y 57.511,Z 215.673,A -85,B 0,C 180,E1 -29136.608,E2 -29136.608} C_VEL
LIN {X 0,Y 58.297,Z 215.857,A -85,B 0,C 180,E1 -29146.052,E2 -29146.052} C_VEL
LIN {X 0,Y 60.514,Z 217.252,A -85,B 0,C 180,E1 -29156.621,E2 -29156.621} C_VEL
LIN {X 0,Y 62.888,Z 222.648,A -85,B 0,C 180,E1 -29166.42,E2 -29166.42} C_VEL
LIN {X 0,Y 64.805,Z 227,A -85,B 0,C 180,E1 -29172.53,E2 -29172.53} C_VEL
LIN {X 0,Y 65.851,Z 229.183,A -85,B 0,C 180,E1 -29175.27,E2 -29175.27} C_VEL
LIN {X 0,Y 67.242,Z 236.241,A -85,B 0,C 180,E1 -29181.461,E2 -29181.461} C_VEL
LIN {X 0,Y 68.383,Z 243.826,A -85,B 0,C 180,E1 -29187.551,E2 -29187.551} C_VEL
LIN {X 0,Y 68.503,Z 247.261,A -85,B 0,C 180,E1 -29190.013,E2 -29190.013} C_VEL
LIN {X 0,Y 66.208,Z 257.123,A -85,B 0,C 180,E1 -29195.965,E2 -29195.965} C_VEL
LIN {X 0,Y 63.311,Z 267.746,A -85,B 0,C 180,E1 -29203.819,E2 -29203.819} C_VEL
LIN {X 0,Y 61.464,Z 271.325,A -85,B 0,C 180,E1 -29206.682,E2 -29206.682} C_VEL
LIN {X 0,Y 56,Z 280.242,A -85,B 0,C 180,E1 -29215.617,E2 -29215.617} C_VEL
LIN {X 0,Y 51.967,Z 287.387,A -85,B 0,C 180,E1 -29226.065,E2 -29226.065} C_VEL
LIN {X 0,Y 49.859,Z 293.136,A -85,B 0,C 180,E1 -29237.795,E2 -29237.795} C_VEL
LIN {X 0,Y 49.53,Z 297.603,A -85,B 0,C 180,E1 -29250.001,E2 -29250.001} C_VEL
LIN {X 0,Y 49.488,Z 299.832,A -85,B 0,C 180,E1 -29258.166,E2 -29258.166} C_VEL
LIN {X 0,Y 51.619,Z 302.972,A -85,B 0,C 180,E1 -29274.11,E2 -29274.11} C_VEL
LIN {X 0,Y 57.204,Z 304.683,A -85,B 0,C 180,E1 -29287.902,E2 -29287.902} C_VEL
LIN {X 0,Y 65.709,Z 305.126,A -85,B 0,C 180,E1 -29298.479,E2 -29298.479} C_VEL
LIN {X 0,Y 76.023,Z 304.276,A -85,B 0,C 180,E1 -29306.308,E2 -29306.308} C_VEL
LIN {X 0,Y 87.453,Z 302.081,A -85,B 0,C 180,E1 -29312.13,E2 -29312.13} C_VEL
LIN {X 0,Y 99.721,Z 298.512,A -85,B 0,C 180,E1 -29316.379,E2 -29316.379} C_VEL
LIN {X 0,Y 101.405,Z 297.635,A -85,B 0,C 180,E1 -29319.723,E2 -29319.723} C_VEL
LIN {X 0,Y 101.728,Z 297.353,A -85,B 0,C 180,E1 -29321.885,E2 -29321.885} C_VEL
LIN {X 0,Y 94.895,Z 299.18,A -85,B 0,C 180,E1 -29324.325,E2 -29324.325} C_VEL
LIN {X 0,Y 86.291,Z 300.94,A -85,B 0,C 180,E1 -29327.787,E2 -29327.787} C_VEL
LIN {X 0,Y 78.061,Z 301.947,A -85,B 0,C 180,E1 -29332.044,E2 -29332.044} C_VEL
LIN {X 0,Y 67.157,Z 302.075,A -85,B 0,C 180,E1 -29339.997,E2 -29339.997} C_VEL
LIN {X 0,Y 61.02,Z 301.363,A -85,B 0,C 180,E1 -29346.61,E2 -29346.61} C_VEL
LIN {X 0,Y 55.81,Z 299.948,A -85,B 0,C 180,E1 -29354.583,E2 -29354.583} C_VEL
LIN {X 0,Y 50.709,Z 296.902,A -85,B 0,C 180,E1 -29367.925,E2 -29367.925} C_VEL
LIN {X 0,Y 48.783,Z 293.696,A -85,B 0,C 180,E1 -29379.18,E2 -29379.18} C_VEL
LIN {X 0,Y 49.17,Z 287.921,A -85,B 0,C 180,E1 -29395.127,E2 -29395.127} C_VEL
LIN {X 0,Y 51.924,Z 281.428,A -85,B 0,C 180,E1 -29407.977,E2 -29407.977} C_VEL
LIN {X 0,Y 55.855,Z 274.428,A -85,B 0,C 180,E1 -29417.94,E2 -29417.94} C_VEL
LIN {X 0,Y 61.137,Z 265.846,A -85,B 0,C 180,E1 -29426.521,E2 -29426.521} C_VEL
LIN {X 0,Y 66.646,Z 256.496,A -85,B 0,C 180,E1 -29433.021,E2 -29433.021} C_VEL
LIN {X 0,Y 69.613,Z 251.169,A -85,B 0,C 180,E1 -29435.793,E2 -29435.793} C_VEL
LIN {X 0,Y 70.057,Z 249.046,A -85,B 0,C 180,E1 -29437.203,E2 -29437.203} C_VEL
LIN {X 0,Y 69.753,Z 243.557,A -85,B 0,C 180,E1 -29441.624,E2 -29441.624} C_VEL
LIN {X 0,Y 68.916,Z 239.375,A -85,B 0,C 180,E1 -29445.302,E2 -29445.302} C_VEL
LIN {X 0,Y 66.992,Z 233.237,A -85,B 0,C 180,E1 -29451.503,E2 -29451.503} C_VEL
LIN {X 0,Y 64.367,Z 227.224,A -85,B 0,C 180,E1 -29459.139,E2 -29459.139} C_VEL
LIN {X 0,Y 63.597,Z 225.237,A -85,B 0,C 180,E1 -29461.816,E2 -29461.816} C_VEL
LIN {X 0,Y 61.499,Z 221.559,A -85,B 0,C 180,E1 -29468.573,E2 -29468.573} C_VEL
LIN {X 0,Y 59.44,Z 217.378,A -85,B 0,C 180,E1 -29478.295,E2 -29478.295} C_VEL
LIN {X 0,Y 57.719,Z 215.813,A -85,B 0,C 180,E1 -29490.857,E2 -29490.857} C_VEL
LIN {X 0,Y 57.511,Z 215.673,A -85,B 0,C 180,E1 -29496.608,E2 -29496.608} C_VEL
LIN {X 0,Y 57.575,Z 215.985,A -85,B 0,C 180,E1 -29500.521,E2 -29500.521} C_VEL
LIN {X 0,Y 57.68,Z 217.655,A -85,B 0,C 180,E1 -29506.19,E2 -29506.19} C_VEL
LIN {X 0,Y 57.772,Z 220.271,A -85,B 0,C 180,E1 -29511.547,E2 -29511.547} C_VEL
LIN {X 0,Y 59.322,Z 228.844,A -85,B 0,C 180,E1 -29525.377,E2 -29525.377} C_VEL
